						arrCyCtrl[arrCyNo.ElectValveName.CaDTCarryingVacuum].Cmd.bON:=TRUE;//负极叠片搬运真空破
						arrCyCtrl[arrCyNo.ElectValveName.CaDTCarryingVacuum].Cmd.bOFF:=FALSE;//负极叠片搬运真空破
						arrCyCtrl[arrCyNo.ElectValveName.CaCarryingVacuum2].Cmd.bON:=TRUE;//负极送片搬运真空破
						arrCyCtrl[arrCyNo.ElectValveName.CaCarryingVacuum2].Cmd.bOFF:=FALSE;//负极送片搬运真空破
						arrCyCtrl[arrCyNo.ElectValveName.CadeviationVacuum].Cmd.bON:=TRUE;//负极纠偏平台真空开
						arrCyCtrl[arrCyNo.ElectValveName.CadeviationVacuum].Cmd.bOFF:=FALSE;//负极纠偏平台真空开			
				
						  Mach_Control.Ca_b.Ca_DPCarryingFalg :=FALSE;//复位负极叠片搬运吸盘上有料标记
						//IF Mach_Control.Ca_b.Ca_CarryingFalg THEN
							Mach_Control.Ca_b.Ca_deviationFalg:=TRUE;//置位纠偏平台上有料标记
							Mach_Control.Ca_b.Ca_CarryingFalg:=FALSE;//复位负极送片搬运吸盘上有料标记
						//END_IF
						Par.stDT_date.Ca_MQ_Slice[8]:=Par.stDT_date.Ca_MQ_Slice[7];
			  END_IF
					
	END_IF	

		
	IF 	arrAxisCtrl[AxiseNo.VirAxisName.VirMain].Status.fActPos>=339   THEN//198
		    IF   NOT An_OverNGMark THEN	
					IF NOT Ca_Number    THEN
						CCD.Over.Start.iPhotoDo:=1;
					ELSE
						CCD.Over.Start.iPhotoDo:=2;
					END_IF
					CCD.Over.Finish.OverhandResult:=0;
					Mach_Control.DT_b.CDD_OverStart:=TRUE;
			  END_IF
					DP_Step3:=121;
					
	END_IF	
121:
	IF 	arrAxisCtrl[AxiseNo.VirAxisName.VirMain].Status.fActPos>=360 THEN//198
		 IF NOT An_OverNGMark THEN	
				arrCyCtrl[arrCyNo.ElectValveName.CaCarryingVacuum2].Cmd.bON:=FALSE;//负极送片搬运真空开
				arrCyCtrl[arrCyNo.ElectValveName.CaCarryingVacuum2].Cmd.bOFF:=TRUE;//负极送片搬运真空开
				arrCyCtrl[arrCyNo.ElectValveName.CaDTCarryingVacuum].Cmd.bON:=FALSE;//负极叠片搬运真空破
				arrCyCtrl[arrCyNo.ElectValveName.CaDTCarryingVacuum].Cmd.bOFF:=TRUE;//负极叠片搬运真空破
		   END_IF	
		DP_Step3:=6666;
	END_IF	
	
	
200://负极叠片，正极在取片位
		IF arrAxisCtrl[AxiseNo.VirAxisName.VirMain].Status.fActPos>=10  AND arrAxisCtrl[AxiseNo.VirAxisName.VirMain].Status.fActPos<=20 THEN//20240508 CF
			An_Step0:=10;//调用正极取片程序
			DP_Step3:=202;		
		END_IF
	
202:
	IF iAnCamInSel2=1 AND NOT An_OverNGMark  THEN
		arrCyCtrl[arrCyNo.ElectValveName.AnDTCarryingVacuum].Cmd.bON:=FALSE;//正极送片搬运真空开
		arrCyCtrl[arrCyNo.ElectValveName.AnDTCarryingVacuum].Cmd.bOFF:=TRUE;//正极送片搬运真空开
	END_IF
	
	//fbAnDTCarryingVacuum.Vacuumsel:=SEL(iAnCamInSel2=1,0,1)     ;//	正极叠片搬运真空开	
	IF arrAxisCtrl[AxiseNo.VirAxisName.VirMain].Status.fActPos>=235 THEN//复检提前
		IF Mach_Control.DT_b.DT_CCD_TwoModel THEN												
			CCD.AnRec.Finish.RectifyResult:=0;
			CCD.AnRec.Finish.RectifyX1:=0;
			CCD.AnRec.Finish.RectifyX2:=0;
			CCD.AnRec.Finish.RectifyY:=0;												
			Mach_Control.An_b.An_CCDStart :=TRUE;//启动CCD拍照
			CCD.AnRec.Start.iPhotoDo:=2;//第二次拍照	
		END_IF
		DP_Step3:=205;
	END_IF
205:			
	IF NOT DP_CheseCam  AND NOT  An_JumpRules[3]  AND NOT  An_JumpRules[6] AND NOT An_JumpRules[8] AND NOT An_JumpRules[10]    THEN
	
				IF arrAxisCtrl[AxiseNo.VirAxisName.VirMain].Status.fActPos>=250  AND arrAxisCtrl[AxiseNo.VirAxisName.VirMain].Status.fActPos<=255 THEN	
					        IF NOT An_OverNGMark THEN
										//fbAnCamInCarryingUpDown.bCamInExecute:=FALSE;//正极升解除耦合															
										//fbAnCamInCarryingWhirling.bCamInExecute:=FALSE;//正极旋转解除耦合			
										//Mach_Control.An_b.An_MainBelting:=FALSE;//正极搬运升降取极片中																					
										IF  NOT  Mach_Control.Ca_b.Ca_deviationFPOK  THEN    //负极放片纠偏太未在初始位置报警  
												Mach_Control.Ca_b.Error_tips[1]:=TRUE ;
										END_IF											
										IF  NOT  Mach_Control.An_b.An_deviationDPOK  THEN    //正极取片纠偏未完成报警
												Mach_Control.An_b.Error_tips[1]:=TRUE;
										END_IF			
										IF Mach_Control.An_b.An_deviationDPOK OR Mach_Control.U.EmptyRunMode OR	TRUE  THEN // 
											arrCyCtrl[arrCyNo.ElectValveName.AnDTCarryingVacuum].Cmd.bON:=FALSE;//正极叠片搬运真空开	
											arrCyCtrl[arrCyNo.ElectValveName.AnDTCarryingVacuum].Cmd.bOFF:=TRUE;//正极叠片搬运真空开		
											An_deviationDPOKFalg:=TRUE;	
										ELSE		
											arrCyCtrl[arrCyNo.ElectValveName.AnDTCarryingVacuum].Cmd.bON:=TRUE;//正极叠片搬运真空关					
											arrCyCtrl[arrCyNo.ElectValveName.AnDTCarryingVacuum].Cmd.bOFF:=FALSE;//正极叠片搬运真空关												
											fbAnCamInDTCarryingUpDown.bCamInExecute:=FALSE;	//正极叠片搬运升降凸轮解耦				
											IF NOT arrAxisCtrl[AxiseNo.AxisName.AnDTCarryingUpDown].Cmd.arrbRealPoint[4]    THEN
													arrAxisCtrl[AxiseNo.AxisName.AnDTCarryingUpDown].Cmd.iGoSetPos:=4;   //到等待位
											END_IF			
										END_IF	
										//IF NOT Mach_Control.An_b.JumpPiceReady THEN
											//An_Step0:=10;//调用正极取片程序	  20240509 CF
										//END_IF
										DP_Step3:=210;				
							 ELSE
							        DP_Step3:=210;	
				             END_IF
				 END_IF			 
	ELSE
									DP_Step3:=210;									
    END_IF

210:
	//打开或关闭真空，标记对应位置有料
	IF 	arrAxisCtrl[AxiseNo.VirAxisName.VirMain].Status.fActPos>=260 THEN//198
		  IF  NOT An_OverNGMark THEN
					CCD.Over.Start.iPliesNo:=UINT_TO_INT(Mach_Control.Ca_b.Ca_Quantited + Mach_Control.An_b.An_Quantited+1);
				    IF (CCD.Over.Start.iPliesNo MOD 2) <>1 OR CCD.Over.Start.iPliesNo=0 THEN
					   Mach_Control.DT_b.Error[69]:=TRUE;//负极对齐度拍照发送层数错误
				    END_IF					
					
					CCD.Over.Start.stPoleNo:=Par.stDT_date.Ca_MQ_Slice[8].stPoleNo;
							Mach_Control.Ca_b.Ca_Rectifydev_CS:=0;
					
							arrCyCtrl[arrCyNo.ElectValveName.CaCarryingVacuum2].Cmd.bON:=TRUE;//负极送片搬运真空关
							arrCyCtrl[arrCyNo.ElectValveName.CaCarryingVacuum2].Cmd.bOFF:=FALSE;//负极送片搬运真空关
							arrCyCtrl[arrCyNo.ElectValveName.CaDTCarryingVacuum].Cmd.bON:=TRUE;//负极叠片搬运直空关
							arrCyCtrl[arrCyNo.ElectValveName.CaDTCarryingVacuum].Cmd.bOFF:=FALSE;//负极叠片搬运直空关
							arrCyCtrl[arrCyNo.ElectValveName.CadeviationVacuum].Cmd.bON:=TRUE;//负极纠偏平台真空开	
							arrCyCtrl[arrCyNo.ElectValveName.CadeviationVacuum].Cmd.bOFF:=FALSE;//负极纠偏平台真空开		
							
							Mach_Control.Ca_b.Ca_DPCarryingFalg :=FALSE;//复位负极叠片搬运吸盘上有料标记
							//IF Mach_Control.Ca_b.Ca_CarryingFalg THEN
								Mach_Control.Ca_b.Ca_deviationFalg:=TRUE;//置位纠偏平台上有料标记
								Mach_Control.Ca_b.Ca_CarryingFalg:=FALSE;//复位负极送片搬运吸盘上有料标记
							//END_IF
							Par.stDT_date.Ca_MQ_Slice[8]:=Par.stDT_date.Ca_MQ_Slice[7];
							IF An_deviationDPOKFalg AND  iAnCamInSel2=1   THEN
									Par.stDT_date.An_MQ_Slice[2]:=Par.stDT_date.An_MQ_Slice[1];
									//IF Mach_Control.An_b.An_deviationFalg THEN
										Mach_Control.An_b.An_DPCarryingFalg :=TRUE;//复位正极叠片搬运吸盘上有料标记										
										Mach_Control.An_b.An_deviationFalg:=FALSE;//置位纠偏平台上有料标记	
									//END_IF										
									arrCyCtrl[arrCyNo.ElectValveName.AndeviationVacuum].Cmd.bOFF:=TRUE;//正极纠偏平台真空关
									arrCyCtrl[arrCyNo.ElectValveName.AndeviationVacuum].Cmd.bON:=FALSE;//正极纠偏平台真空关
									arrCyCtrl[arrCyNo.ElectValveName.AndeviationVacuumBark].Cmd.bON:=TRUE;//正极纠偏平台破真空开	
									arrCyCtrl[arrCyNo.ElectValveName.AndeviationVacuumBark].Cmd.bOFF:=FALSE;//正极纠偏平台破真空开	
							 END_IF			
							(*	
								ELSIF NOT   DP_CheseCam THEN								
									An_Step3:=10;//正极叠片搬运取纠偏台极片	
							*)																					
	        END_IF
				 
				 
	END_IF
	
	IF 	arrAxisCtrl[AxiseNo.VirAxisName.VirMain].Status.fActPos>=339 THEN//198
		  IF  NOT An_OverNGMark THEN
				IF NOT Ca_Number  THEN
					CCD.Over.Start.iPhotoDo:=1;
				ELSE
					CCD.Over.Start.iPhotoDo:=2;
				END_IF
				CCD.Over.Finish.OverhandResult:=0;
				Mach_Control.DT_b.CDD_OverStart:=TRUE;			
	       END_IF
				 
			IF NOT Ca_Number THEN
				DP_Step3:=211;					
			END_IF
	END_IF
	

211:
	IF 	arrAxisCtrl[AxiseNo.VirAxisName.VirMain].Status.fActPos>=360 THEN//198	
		 IF NOT An_OverNGMark THEN	
				arrCyCtrl[arrCyNo.ElectValveName.CaCarryingVacuum2].Cmd.bON:=FALSE;//负极送片搬运真空开
				arrCyCtrl[arrCyNo.ElectValveName.CaCarryingVacuum2].Cmd.bOFF:=TRUE;//负极送片搬运真空开
				arrCyCtrl[arrCyNo.ElectValveName.CaDTCarryingVacuum].Cmd.bON:=FALSE;//负极叠片搬运直空开
				arrCyCtrl[arrCyNo.ElectValveName.CaDTCarryingVacuum].Cmd.bOFF:=TRUE;//负极叠片搬运直空开
		END_IF		
		DP_Step3:=6666;					
	END_IF
			



		
300://正极叠片，负极在取片位			
	bStandbyStep1_3:=FALSE;
	bStandbyStep1_4:=FALSE;
	DP_Step3:=310; 		
310:	
	IF arrAxisCtrl[AxiseNo.VirAxisName.VirMain].Status.fActPos>=10  AND  arrAxisCtrl[AxiseNo.VirAxisName.VirMain].Status.fActPos<=245    THEN
		//正送片搬运极取片处理
		IF   arrAxisCtrl[AxiseNo.AxisName.CaCarryingUpDown2].Cmd.arrbRealPoint[4] AND 
			NOT Mach_Control.Ca_b.Ca_CarryingFalg    AND  ( Mach_Control.Ca_b.Ca_CacheBeltDLOK OR  Mach_Control.U.EmptyRunMode )  AND 
			NOT  Mach_Control.Ca_b.Ca_CacheBelting   AND NOT  bStandbyStep1_3 	 THEN
			Ca_Step0:=10;   //负极取流水线子程序
			bStandbyStep1_3:=TRUE;
		END_IF
	
		IF arrAxisCtrl[AxiseNo.AxisName.CaDTCarryingUpDown].Cmd.arrbRealPoint[4] AND 
			Mach_Control.Ca_b.Ca_deviationDPOK AND NOT Mach_Control.Ca_b.Ca_DPCarryingFalg AND  
			Mach_Control.Ca_b.Ca_deviationFalg AND  NOT  bStandbyStep1_4   
           AND   NOT Ca_OverNGMark THEN
			Ca_Step3:=10;     //负极取纠偏平台子程序
			bStandbyStep1_4:=TRUE;
		END_IF					
	ELSIF  arrAxisCtrl[AxiseNo.VirAxisName.VirMain].Status.fActPos>245  THEN
		    IF  NOT Ca_OverNGMark THEN
			      DP_Step3:=320; 
			ELSE	  
				  DP_Step3:=6666;	
			END_IF		  
	END_IF	
	
320://正极叠片，负极在取片位
   IF NOT Ca_OverNGMark THEN
		arrCyCtrl[arrCyNo.ElectValveName.AndeviationVacuum].Cmd.bON:=TRUE;//正极纠偏平台真空开			
		arrCyCtrl[arrCyNo.ElectValveName.AndeviationVacuum].Cmd.bOFF:=FALSE;//正极纠偏平台真空开		
	END_IF					
	IF 	arrAxisCtrl[AxiseNo.VirAxisName.VirMain].Status.fActPos>=260 THEN//198

		IF NOT Ca_OverNGMark THEN
				CCD.Over.Start.iPliesNo:=UINT_TO_INT(Mach_Control.Ca_b.Ca_Quantited + Mach_Control.An_b.An_Quantited+1);
				    IF (CCD.Over.Start.iPliesNo MOD 2) <>0 OR CCD.Over.Start.iPliesNo=0 THEN
					   Mach_Control.DT_b.Error[68]:=TRUE;//正极对齐度拍照发送层数错误
				    END_IF				
				
				CCD.Over.Start.stPoleNo:=Par.stDT_date.An_MQ_Slice[2].stPoleNo;
				Mach_Control.An_b.An_Rectifydev_CS:=0;				
		
				arrCyCtrl[arrCyNo.ElectValveName.AnCarryingVacuum].Cmd.bON:=FALSE;//正极送片搬运真空关
				arrCyCtrl[arrCyNo.ElectValveName.AnCarryingVacuum].Cmd.bOFF:=TRUE;//正极送片搬运真空关
				arrCyCtrl[arrCyNo.ElectValveName.AnCarryingVacuumBark].Cmd.bON:=TRUE;//正极送片搬运破真空开
				arrCyCtrl[arrCyNo.ElectValveName.AnCarryingVacuumBark].Cmd.bOFF:=FALSE;//正极送片搬运破真空开
				
				arrCyCtrl[arrCyNo.ElectValveName.AnDTCarryingVacuum].Cmd.bON:=TRUE;//正极送片搬运真空关
				arrCyCtrl[arrCyNo.ElectValveName.AnDTCarryingVacuum].Cmd.bOFF:=FALSE;//正极送片搬运真空关
				//arrCyCtrl[arrCyNo.ElectValveName.AnDTCarryingVacuumBark].Cmd.bON:=TRUE;//正极送片搬运破真空开
				//arrCyCtrl[arrCyNo.ElectValveName.AnDTCarryingVacuumBark].Cmd.bOFF:=FALSE;//正极送片搬运破真空开
				
				arrCyCtrl[arrCyNo.ElectValveName.AndeviationVacuum].Cmd.bON:=TRUE;//正极纠偏平台真空开		
				arrCyCtrl[arrCyNo.ElectValveName.AndeviationVacuum].Cmd.bOFF:=FALSE;//正极纠偏平台真空开		
				
				
				Mach_Control.An_b.An_DPCarryingFalg :=FALSE;//复位正极叠片搬运吸盘上有料标记
				//IF Mach_Control.An_b.An_CarryingFalg THEN
					Mach_Control.An_b.An_deviationFalg:=TRUE;//置位纠偏平台上有料标记
					Mach_Control.An_b.An_CarryingFalg:=FALSE;//复位正极送片搬运吸盘上有料标记
				//END_IF
				Par.stDT_date.An_MQ_Slice[1]:=Par.stDT_date.An_MQ_Slice[0];
	      END_IF				
	 END_IF

	IF 	arrAxisCtrl[AxiseNo.VirAxisName.VirMain].Status.fActPos>=339 THEN//198
		   IF NOT Ca_OverNGMark THEN
				IF NOT An_Number  THEN
					CCD.Over.Start.iPhotoDo:=1;
				ELSE
					CCD.Over.Start.iPhotoDo:=2;
				END_IF
				CCD.Over.Finish.OverhandResult:=0;
				Mach_Control.DT_b.CDD_OverStart:=TRUE;	
	       END_IF      
		  DP_Step3:=6666;	
	END_IF	
			

400:	//复检提前------//正极叠片，负极在叠片位
		IF arrAxisCtrl[AxiseNo.VirAxisName.VirMain].Status.fActPos>=10  AND arrAxisCtrl[AxiseNo.VirAxisName.VirMain].Status.fActPos<=20 THEN//20240508 CF																			
			Ca_Step0:=10;//调用负极取片程序       取片允许条件在子程序里
			DP_Step3:=402;
		END_IF

402:	
	//fbCaDTCarryingVacuum.Vacuumsel:= SEL(iCaCamInSel2=1 ,0,1)   ;//	负极叠片搬运真空开
	IF iCaCamInSel2=1 AND NOT Ca_OverNGMark THEN
		arrCyCtrl[arrCyNo.ElectValveName.CaDTCarryingVacuum].Cmd.bON:=FALSE;//负极叠台搬运真空开	
		arrCyCtrl[arrCyNo.ElectValveName.CaDTCarryingVacuum].Cmd.bOFF:=TRUE;//负极叠台搬运真空开		
	END_IF

	IF 	arrAxisCtrl[AxiseNo.VirAxisName.VirMain].Status.fActPos>=235 THEN//198
		IF Mach_Control.DT_b.DT_CCD_TwoModel THEN
				CCD.CaRec.Finish.RectifyX1:=0;
				CCD.CaRec.Finish.RectifyX2:=0;
				CCD.CaRec.Finish.RectifyY:=0;		
				CCD.CaRec.Finish.RectifyResult:=0;//拍照结果清零									
				Mach_Control.Ca_b.Ca_CCDStart :=TRUE;//启动CCD拍照
				CCD.CaRec.Start.iPhotoDo:=2;//启动CCD第二次拍照									
		END_IF
		DP_Step3:=405;
	END_IF
405:		
 
				IF arrAxisCtrl[AxiseNo.VirAxisName.VirMain].Status.fActPos>=250  AND arrAxisCtrl[AxiseNo.VirAxisName.VirMain].Status.fActPos<=255 THEN		
						  IF  NOT Ca_OverNGMark	  THEN															
										IF  NOT  Mach_Control.An_b.An_deviationFPOK  THEN    //正极放片纠偏太未在初始位置报警  
											  Mach_Control.An_b.Error_tips[2]:=TRUE ;
										END_IF
										
										IF  NOT  Mach_Control.Ca_b.Ca_deviationDPOK  THEN    //负极取片纠偏未完成报警
											  Mach_Control.Ca_b.Error_tips[2]:=TRUE ;
										END_IF		
								
										//正极叠片时平移到位后判断正极纠偏台是否允许放片
										IF Mach_Control.An_b.An_deviationFPOK OR Mach_Control.U.EmptyRunMode  THEN 
												An_deviationFPOKFalg:=TRUE;//正极纠偏平台允许放片标记
										ELSE									
											fbAnCamInCarryingUpDown.bCamInExecute:=FALSE;	//正极送片搬运升降凸轮解耦				
											IF NOT arrAxisCtrl[AxiseNo.AxisName.AnCarryingUpDown].Cmd.arrbRealPoint[4]    THEN
												arrAxisCtrl[AxiseNo.AxisName.AnCarryingUpDown].Cmd.iGoSetPos:=4;
											END_IF;				
										END_IF					
										IF Mach_Control.Ca_b.Ca_deviationDPOK OR Mach_Control.U.EmptyRunMode OR TRUE  THEN //  
											Ca_deviationDPOKFalg:=TRUE;	
											arrCyCtrl[arrCyNo.ElectValveName.CaDTCarryingVacuum].Cmd.bON:=FALSE;//负极叠片搬运真空开	
											arrCyCtrl[arrCyNo.ElectValveName.CaDTCarryingVacuum].Cmd.bOFF:=TRUE;//负极叠片搬运真空开		
										ELSE	
											//arrCyCtrl[arrCyNo.ElectValveName.CaDTCarryingVacuum].Cmd.bON:=FALSE;//负极叠片搬运真空开									
											fbCaCamInDTCarryingUpDown.bCamInExecute:=FALSE;	//负极叠片搬运升降凸轮解耦				
											IF NOT arrAxisCtrl[AxiseNo.AxisName.CaDTCarryingUpDown].Cmd.arrbRealPoint[4]    THEN
												arrAxisCtrl[AxiseNo.AxisName.CaDTCarryingUpDown].Cmd.iGoSetPos:=4;   //到等待位
											ELSE
												arrAxisCtrl[AxiseNo.AxisName.CaDTCarryingUpDown].Cmd.iGoSetPos:=0;   //到等待位
											END_IF;				
										END_IF			
											//Ca_Step0:=10;//调用负极取片程序       取片允许条件在子程序里 20240509 CF
											DP_Step3:=410;	
							ELSE
										   DP_Step3:=6666;			
							END_IF									
									
	           END_IF
	
(*	
	//判断是否允许负极送片搬运取料
	IF arrAxisCtrl[AxiseNo.VirAxisName.VirMain].Status.fActPos>=CamOutArgel  AND arrAxisCtrl[AxiseNo.VirAxisName.VirMain].Status.fActPos<=(CamOutArgel+5) THEN
		IF (Mach_Control.Ca_b.Ca_CacheBeltDLOK AND NOT fbCaCamInCarryingUpDown2OutCamFlge) OR Mach_Control.U.EmptyRunMode  THEN
			Mach_Control.Ca_b.Ca_CacheBelting:=TRUE;//f负极搬运升降取极片中	
			arrCyCtrl[arrCyNo.ElectValveName.CaCarryingVacuum2].Cmd.bON:=FALSE;//负极送片搬运真空开
			arrCyCtrl[arrCyNo.ElectValveName.CaCarryingVacuum2].Cmd.bOFF:=TRUE;//负极送片搬运真空开
		ELSE
			//arrCyCtrl[arrCyNo.ElectValveName.CaCarryingVacuum2].Cmd.bON:=FALSE;//负极送片搬运真空开
			fbCaCamInCarryingUpDown2.bCamInExecute:=FALSE;//负极升解除耦合
			Mach_Control.Ca_b.Ca_CacheBelting:=FALSE;
		END_IF								
	END_IF
	//解除负极搬运升降凸轮耦合标记
	fbCaCamInCarryingUpDown2OutCam_F_TRIG(CLK:=fbCaCamInCarryingUpDown2.bCamInExecute , Q=> );
	IF fbCaCamInCarryingUpDown2OutCam_F_TRIG.Q THEN
		fbCaCamInCarryingUpDown2OutCamFlge:=TRUE;//负极升降2凸轮解耦标记
	END_IF	
*)			
410:							
	//打开或关闭真空，标记对应位置有料
	IF 	arrAxisCtrl[AxiseNo.VirAxisName.VirMain].Status.fActPos>=260 THEN//198
		CCD.Over.Start.iPliesNo:=UINT_TO_INT(Mach_Control.Ca_b.Ca_Quantited + Mach_Control.An_b.An_Quantited+1);	
		IF (CCD.Over.Start.iPliesNo MOD 2) <>0 OR CCD.Over.Start.iPliesNo=0 THEN
		   Mach_Control.DT_b.Error[68]:=TRUE;//正极对齐度拍照发送层数错误
		END_IF	
	
		Mach_Control.An_b.An_Rectifydev_CS:=0;
			
					CCD.Over.Start.stPoleNo:=Par.stDT_date.An_MQ_Slice[2].stPoleNo;
				(*	
					arrCyCtrl[arrCyNo.ElectValveName.AnCarryingVacuum].Cmd.bOFF:=TRUE;//正极送片搬运真空关
					arrCyCtrl[arrCyNo.ElectValveName.AnCarryingVacuumBark].Cmd.bON:=TRUE;//正极送片搬运破真空开
					arrCyCtrl[arrCyNo.ElectValveName.AnDTCarryingVacuum].Cmd.bOFF:=TRUE;//正极叠片搬运真空关
					arrCyCtrl[arrCyNo.ElectValveName.AnDTCarryingVacuumBark].Cmd.bON:=TRUE;//正极叠片搬运破真空开
				*)	
					arrCyCtrl[arrCyNo.ElectValveName.AnCarryingVacuum].Cmd.bON:=FALSE;//正极送片搬运真空关
					arrCyCtrl[arrCyNo.ElectValveName.AnCarryingVacuum].Cmd.bOFF:=TRUE;//正极送片搬运真空关
					arrCyCtrl[arrCyNo.ElectValveName.AnCarryingVacuumBark].Cmd.bON:=TRUE;//正极送片搬运破真空开
					arrCyCtrl[arrCyNo.ElectValveName.AnCarryingVacuumBark].Cmd.bOFF:=FALSE;//正极送片搬运破真空开
					
					arrCyCtrl[arrCyNo.ElectValveName.AnDTCarryingVacuum].Cmd.bON:=TRUE;//正极送片搬运真空关
					arrCyCtrl[arrCyNo.ElectValveName.AnDTCarryingVacuum].Cmd.bOFF:=FALSE;//正极送片搬运真空关
					//arrCyCtrl[arrCyNo.ElectValveName.AnDTCarryingVacuumBark].Cmd.bON:=TRUE;//正极送片搬运破真空开
				//	arrCyCtrl[arrCyNo.ElectValveName.AnDTCarryingVacuumBark].Cmd.bOFF:=FALSE;//正极送片搬运破真空开	
					
					arrCyCtrl[arrCyNo.ElectValveName.AndeviationVacuum].Cmd.bON:=TRUE;//正极纠偏平台真空开	
					arrCyCtrl[arrCyNo.ElectValveName.AndeviationVacuum].Cmd.bOFF:=FALSE;//正极纠偏平台真空开	
			
					Mach_Control.An_b.An_DPCarryingFalg :=FALSE;//复位正极叠片搬运吸盘上有料标记
					//IF Mach_Control.An_b.An_CarryingFalg THEN
						Mach_Control.An_b.An_deviationFalg:=TRUE;//置位纠偏平台上有料标记
						Mach_Control.An_b.An_CarryingFalg:=FALSE;//复位正极送片搬运吸盘上有料标记
					//END_IF
					
					Par.stDT_date.An_MQ_Slice[1]:=Par.stDT_date.An_MQ_Slice[0];
					
					(*
					IF (Mach_Control.Ca_b.Ca_CacheBelting AND NOT fbCaCamInCarryingUpDown2OutCamFlge) OR Mach_Control.U.EmptyRunMode  THEN
						Mach_Control.Ca_b.Ca_CarryingFalg:=TRUE;//复位负极送片搬运吸盘上有料标记
						Par.stDT_date.Ca_MQ_Slice[7]:=Par.stDT_date.Ca_MQ_Slice[6];
					END_IF*)
					
					
					arrAxisCtrl[AxiseNo.AxisName.CaCarryingUpDown2].Cmd.bStop:=FALSE;
				


		//判断负极纠偏台是否允许取料
		IF Ca_deviationDPOKFalg AND NOT DP_CheseCam AND iCaCamInSel2=1 AND   NOT Ca_OverNGMark	 THEN		
			arrCyCtrl[arrCyNo.ElectValveName.CaDTCarryingVacuum].Cmd.bON:=FALSE;//负极叠台搬运真空开	
			arrCyCtrl[arrCyNo.ElectValveName.CaDTCarryingVacuum].Cmd.bOFF:=TRUE;//负极叠台搬运真空开	
			arrCyCtrl[arrCyNo.ElectValveName.CadeviationVacuum].Cmd.bOFF:=TRUE;//负极纠偏平台真空关
			arrCyCtrl[arrCyNo.ElectValveName.CadeviationVacuum].Cmd.bON:=FALSE;//负极纠偏平台真空关
			arrCyCtrl[arrCyNo.ElectValveName.CadeviationVacuumBark].Cmd.bON:=TRUE;//负极纠偏平台破真空开	
			arrCyCtrl[arrCyNo.ElectValveName.CadeviationVacuumBark].Cmd.bOFF:=FALSE;//负极纠偏平台破真空开		
			//IF 	Mach_Control.Ca_b.Ca_deviationFalg THEN				
				Mach_Control.Ca_b.Ca_DPCarryingFalg :=TRUE;//置位负极叠片搬运吸盘上有料标记			
				Mach_Control.Ca_b.Ca_deviationFalg:=FALSE;//复位负极纠偏平台上有料标记	
			//END_IF			
			Par.stDT_date.Ca_MQ_Slice[9]:=Par.stDT_date.Ca_MQ_Slice[8];
		(*	
		ELSE   
			Ca_Step3:=10;//负极叠片搬运取纠偏台极片	
		*)	   
		END_IF									

		//判断正极纠偏台是否允许放料
		IF  NOT Ca_OverNGMark	 THEN		
				IF An_deviationFPOKFalg THEN			
					arrCyCtrl[arrCyNo.ElectValveName.AnCarryingVacuumBark].Cmd.bON:=TRUE;//正极送片搬运真空关
					arrCyCtrl[arrCyNo.ElectValveName.AnCarryingVacuumBark].Cmd.bOFF:=FALSE;//正极送片搬运破真空开
					arrCyCtrl[arrCyNo.ElectValveName.AndeviationVacuum].Cmd.bON:=TRUE;//正极纠偏平台真空开		
					arrCyCtrl[arrCyNo.ElectValveName.AndeviationVacuum].Cmd.bOFF:=FALSE;//正极纠偏平台真空开	
					//IF Mach_Control.An_b.An_CarryingFalg THEN	
						Mach_Control.An_b.An_deviationFalg:=TRUE;//置位正极纠偏平台上有料标记
						Mach_Control.An_b.An_CarryingFalg:=FALSE;//复位正极送片搬运吸盘上有料标记						
					//END_IF			
					Par.stDT_date.An_MQ_Slice[1]:=Par.stDT_date.An_MQ_Slice[0];//送片机械手传送至纠偏平台
					ELSE   
						An_Step1:=10;//正极送片搬运放片到纠偏台			   
					END_IF
			END_IF 
	END_IF

	IF 	arrAxisCtrl[AxiseNo.VirAxisName.VirMain].Status.fActPos>=339 THEN//198
		 IF NOT Ca_OverNGMark THEN
				IF NOT An_Number THEN
					CCD.Over.Start.iPhotoDo:=1;
				ELSE
					CCD.Over.Start.iPhotoDo:=2;
				END_IF
				CCD.Over.Finish.OverhandResult:=0;
				Mach_Control.DT_b.CDD_OverStart:=TRUE;	
	    END_IF
			
		IF NOT An_Number THEN
			DP_Step3:=6666;					
		END_IF

	
	END_IF
	

END_CASE



//判断主轴是否完成
CASE  DP_Step4 OF
100://叠负极主轴定位完成判断	
		//叠负极主轴在当前周期220度之前对齐度NG为上一片结果
      IF (((arrAxisCtrl[AxiseNo.VirAxisName.VirMain].Status.fActPos>10 AND  arrAxisCtrl[AxiseNo.VirAxisName.VirMain].Status.fActPos<230) AND 
           (CCD.Over.Finish.OverhandResult=2 OR  CCD.Over.Finish.OverhandResult=3 OR CCD.Over.Finish.OverhandResult=4 ) ) OR
		  (arrAxisCtrl[AxiseNo.VirAxisName.VirMain].Status.fActPos>=230 AND  arrAxisCtrl[AxiseNo.VirAxisName.VirMain].Status.fActPos<235 AND 
           CCD.Over.Finish.OverhandResult=0  ))  AND
           NOT Mach_Control.DT_b.DT_Overhang AND  NOT  Mach_Control.U.EmptyRunMode AND NOT Mach_Control.DT_b.DT_Sheetkick AND  
           Mach_Control.Ca_b.Ca_Quantited>0  AND NOT Ca_OverNGMark AND NOT OversequelNG AND NOT Bnt_Blueflaging THEN
		  An_OverNGMark:=TRUE;//上一片正极对齐度NG标记
	  END_IF

	  
	 IF  arrAxisCtrl[AxiseNo.VirAxisName.VirMain].Status.fActPos>240  THEN 
	      Ca_OverNGMark:=FALSE;
	  END_IF
	   
	IF arrAxis[AxiseNo.VirAxisName.VirMain].NcToPlc.SetPos=360 AND  arrAxis[AxiseNo.VirAxisName.VirMain].Status.NotMoving  THEN
		//如果，叠片搬运掉片报警就不计数		
		IF NOT Ca_Number AND NOT An_OverNGMark THEN
						Mach_Control.Ca_b.Ca_Quantited:=Mach_Control.Ca_b.Ca_Quantited+1;
						DPcount:=DPcount+1;
						IF Mach_Control.U.EmptyRunMode THEN
							Mach_Control.Ca_b.Ca_EmptyRunKDQuantited:=Mach_Control.Ca_b.Ca_EmptyRunKDQuantited +1;
						//			ELSE
						//				Mach_Control.Ca_b.Ca_EmptyRunKDQuantited:=0;
						END_IF
						Par.stDT_date.YD_JS_L:=Par.stDT_date.YD_JS_L+1;
						Par.stDT_date.YD_ferrJS:=Par.stDT_date.YD_ferrJS+1;
						Mach_Control.Ca_b.Ca_CCD_amount:=0;
							//叠台升降轴下降
							IF NOT Mach_Control.U.EmptyRunMode  THEN
								arrAxisCtrl[AxiseNo.AxisName.DTUpDown].Cmd.fPosition_of_Rel:=-(Par.stDT_date.Ca_Thickness+Par.stDT_date.SEPTA_Thickness+Par.stDT_date.Pole_ThicknessCom);
							ELSE
								arrAxisCtrl[AxiseNo.AxisName.DTUpDown].Cmd.fPosition_of_Rel:=-Par.stDT_date.SEPTA_Thickness;
							END_IF
							IF Mach_Control.Ca_b.Ca_Quantited + Mach_Control.An_b.An_Quantited>3 THEN
								arrAxisPar[AxiseNo.AxisName.DTUpDown].fVelocity_of_Rel:=100;
								arrAxisCtrl[AxiseNo.AxisName.DTUpDown].Cmd.bMoveRel:=TRUE;
							END_IF
		END_IF
		Mach_Control.An_b.An_CCDStart :=FALSE;//启动CCD拍照						
		DP_Step1:=100;//解除耦合，主轴回零子程序
	    

		IF Mach_Control.DT_b.SinStepMode THEN//单步调试模式
			DP_SinStepe:=TRUE;
		ELSE
			DP_SinStepe:=FALSE;	
		END_IF
		
		//DP_Step0:=0;
		Ca_AlarmTON[11].IN:=FALSE;
		IF Ca_Number  OR An_OverNGMark THEN
			DP_Step6:=6666;
		ELSIF Mach_Control.DT_b.DT_Overhang THEN
			DP_Step6:=102;
		ELSE
			DP_Step6:=101;
		END_IF	
		DP_Step4:=110;
        DPtime:=10;	
	END_IF;	
110:
	IF ((*Ca_deviationFPOKFalg OR*) Ca_Step1=6666 OR Ca_Step1=0) AND ((*An_deviationDPOKFalg OR *)An_Step3=6666 OR An_Step3=0)  
		AND ((An_Step0=6666 OR An_Step0=0) OR Mach_Control.An_b.An_Quantited=Par.stDT_date.An_Quantity )  THEN         
		DP_Step4:=6666;
			IF   NOT An_OverNGMark THEN
	        	DP_Step0:=0;
				DPtime:=11;	
		       Ca_deviationFPOKFalg:=FALSE;
		       An_deviationDPOKFalg:=FALSE;  
			ELSE   
			    DP_Step0:=10;
		     	An_OverNGStep:=1000;	//踢正极对齐度NG片
				 CCD.Over.Finish.OverhandResult:=0;	
	       END_IF;				
	END_IF



		
200:	//叠正极主轴定位完成判断
	  //叠正极主轴在当前周期220度之前对齐度NG为上一片结果
	   IF (((arrAxisCtrl[AxiseNo.VirAxisName.VirMain].Status.fActPos>10 AND  arrAxisCtrl[AxiseNo.VirAxisName.VirMain].Status.fActPos<230) AND 
           (CCD.Over.Finish.OverhandResult=2 OR  CCD.Over.Finish.OverhandResult=3 OR CCD.Over.Finish.OverhandResult=4 )) OR
           (arrAxisCtrl[AxiseNo.VirAxisName.VirMain].Status.fActPos>=230 AND  arrAxisCtrl[AxiseNo.VirAxisName.VirMain].Status.fActPos<235 AND 
            CCD.Over.Finish.OverhandResult=0))  AND     
           NOT Mach_Control.DT_b.DT_Overhang AND NOT  Mach_Control.U.EmptyRunMode  AND NOT Mach_Control.DT_b.DT_Sheetkick AND
           Mach_Control.Ca_b.Ca_Quantited>0  AND NOT An_OverNGMark AND NOT OversequelNG AND NOT Bnt_Blueflaging THEN
		  Ca_OverNGMark:=TRUE;//上一片负极对齐度NG标记
	  END_IF
	
	 	 IF  arrAxisCtrl[AxiseNo.VirAxisName.VirMain].Status.fActPos>240 THEN 
	      An_OverNGMark:=FALSE;
	  END_IF 
	  
	
	IF arrAxis[AxiseNo.VirAxisName.VirMain].NcToPlc.SetPos=360 AND  arrAxis[AxiseNo.VirAxisName.VirMain].Status.NotMoving  THEN
		//如果，叠片搬运掉片报警就不计数				
		IF NOT An_Number AND NOT Ca_OverNGMark THEN
						Mach_Control.An_b.An_Quantited:=Mach_Control.An_b.An_Quantited+1;
						DPcount:=DPcount+1;			
						IF Mach_Control.U.EmptyRunMode THEN
							Mach_Control.An_b.An_EmptyRunKDQuantited:=Mach_Control.An_b.An_EmptyRunKDQuantited +1;
						//			ELSE
						//				Mach_Control.An_b.An_EmptyRunKDQuantited:=0;
						END_IF
						Par.stDT_date.YD_JS_R:=Par.stDT_date.YD_JS_R+1;
						Mach_Control.An_b.An_CCD_amount:=0;
						//叠台升降轴下降
						IF NOT Mach_Control.U.EmptyRunMode  THEN
								arrAxisCtrl[AxiseNo.AxisName.DTUpDown].Cmd.fPosition_of_Rel:=-(Par.stDT_date.An_Thickness+Par.stDT_date.SEPTA_Thickness+Par.stDT_date.Pole_ThicknessCom);
						ELSE
								arrAxisCtrl[AxiseNo.AxisName.DTUpDown].Cmd.fPosition_of_Rel:=-Par.stDT_date.SEPTA_Thickness;
						END_IF
						IF Mach_Control.Ca_b.Ca_Quantited + Mach_Control.An_b.An_Quantited>3 THEN
								arrAxisPar[AxiseNo.AxisName.DTUpDown].fVelocity_of_Rel:=100;
								arrAxisCtrl[AxiseNo.AxisName.DTUpDown].Cmd.bMoveRel:=TRUE;
						END_IF	
		END_IF
		Mach_Control.Ca_b.Ca_CCDStart :=FALSE;//启动CCD拍照			
		DP_Step1:=100;//解除耦合，主轴回零	
        
		(*
		IF  (Mach_Control.Ca_b.Ca_CacheBelting AND NOT fbCaCamInCarryingUpDown2OutCamFlge) OR Mach_Control.U.EmptyRunMode  THEN
			Par.stDT_date.Ca_betlCount.5:=FALSE;//复位负极流水线极片标记
			Mach_Control.Ca_b.Ca_CacheBelting:=FALSE;
		END_IF	*)
	
						
		arrCyCtrl[arrCyNo.ElectValveName.CadeviationVacuumBark].Cmd.bOFF:=TRUE;//负极纠偏平台破真空关	
		IF Mach_Control.DT_b.SinStepMode THEN//单步调试模式
			DP_SinStepe:=TRUE;
		ELSE
			DP_SinStepe:=FALSE;	
		END_IF							
		//DP_Step0:=0;
		An_AlarmTON[11].IN:=FALSE;
		IF An_Number OR Ca_OverNGMark THEN
			  DP_Step7:=6666;
		ELSIF  Mach_Control.DT_b.DT_Overhang THEN
			  DP_Step7:=202;
		ELSE
			  DP_Step7:=201;
		END_IF
		DP_Step4:=210;	
		DPtime:=20;	
		(*	
			IF  Mach_Control.DT_b.DT_Overhang AND NOT An_Number THEN
				  DP_Step7:=202;
			ELSIF An_Number THEN
				  DP_Step7:=6666;
			ELSE
				  DP_Step7:=201;
			END_IF
			DP_Step4:=6666;	
		*)
	END_IF;	
210:
	IF ((*An_deviationFPOKFalg OR *)An_Step1=6666 OR An_Step1=0) AND ((*Ca_deviationDPOKFalg OR *)Ca_Step3=6666 OR Ca_Step3=0) 
	AND (Ca_Step0=6666 OR Ca_Step0=0) THEN       
          	DP_Step4:=6666;
          IF NOT Ca_OverNGMark THEN
				DP_Step0:=0;
				DPtime:=21;	
				An_deviationFPOKFalg:=FALSE;
				Ca_deviationDPOKFalg:=FALSE; 
			ELSE	
			    DP_Step0:=20;
		     	Ca_OverNGStep:=1000;	//踢负极对齐度NG片
                CCD.Over.Finish.OverhandResult:=0;	
          END_IF
			
	END_IF

			
END_CASE



//观察NG片用，发现问题后删除
IF Ca_NGTest1.Q THEN
	Ca_NG:=Ca_NG+1;
END_IF


CASE  DP_Step5 OF
100://判断主轴运行时负极叠片搬运升降真空报警
	IF arrAxisCtrl[AxiseNo.VirAxisName.VirMain].Status.fActPos>0 AND arrAxisCtrl[AxiseNo.VirAxisName.VirMain].Status.fActPos<235 THEN
		IF Ca_Number OR An_OverNGMark  THEN	
			IF Ca_Number THEN
				AnOverNGcount:=0; 
				arrCyCtrl[arrCyNo.ElectValveName.CaDTCarryingVacuum].Cmd.bON:=TRUE;//负极叠片搬运破真空开	
				arrCyCtrl[arrCyNo.ElectValveName.CaDTCarryingVacuum].Cmd.bOFF:=FALSE;//负极叠片搬运破真空开	
			END_IF	
				DP_Step5:=110;
		END_IF
		Ca_NGTest1(CLK:=(CCD.CaRec.Finish.RectifyResult=2) , Q=> );
	ELSE
		AnOverNGcount:=0; 
		DP_Step5:=6666;
	END_IF

110://叠负极主轴220度之前有对齐度NG, 负极送片搬运升降、负极叠台搬运升降、右压刀开合、右压刀升降、正极叠台搬运升降轴解耦  ,踢掉上一片正极
	fbCaCamInDTCarryingUpDown.bCamInExecute:=FALSE;//负极叠片搬运升降
	fbCamInLeftYDUpDown.bCamInExecute:=FALSE;//左压刀升降
	fbCamInLeftYDLine.bCamInExecute:=FALSE;//左压刀开合
	IF  An_OverNGMark THEN
		fbCaCamInCarryingUpDown2.bCamInExecute:=FALSE;//负极s送片搬运升降
		fbAnCamInDTCarryingUpDown.bCamInExecute:=FALSE;//正极叠片搬运升降
		IF NOT Mach_Control.An_b.An_DPCarryingFalg THEN
			arrCyCtrl[arrCyNo.ElectValveName.AnDTCarryingVacuum].Cmd.bON:=TRUE;//正极叠片搬运真空真空关
			arrCyCtrl[arrCyNo.ElectValveName.AnDTCarryingVacuum].Cmd.bOFF:=FALSE;//正极叠片搬运真空真空关
		END_IF	
	END_IF
	 
	IF NOT  fbCaCamInDTCarryingUpDown.bCamInExecute AND NOT fbCamInLeftYDUpDown.bCamInExecute AND NOT  fbCamInLeftYDLine.bCamInExecute AND 
        (( NOT  fbCaCamInCarryingUpDown2.bCamInExecute AND NOT  fbAnCamInDTCarryingUpDown.bCamInExecute ) OR NOT An_OverNGMark )   THEN
	       IF Ca_Number THEN
				arrCyCtrl[arrCyNo.ElectValveName.CaDTCarryingVacuum].Cmd.bON:=FALSE;//负极叠片搬运真空开
				arrCyCtrl[arrCyNo.ElectValveName.CaDTCarryingVacuum].Cmd.bOFF:=TRUE;//负极叠片搬运真空开
			END_IF	
			DP_Step5:=120;
	END_IF

120:
	arrAxisCtrl[AxiseNo.AxisName.CaDTCarryingUpDown].Cmd.bGearOut:=TRUE;
	arrAxisCtrl[AxiseNo.AxisName.LeftYDLine].Cmd.bGearOut:=TRUE;
	arrAxisCtrl[AxiseNo.AxisName.LeftYDUpDown].Cmd.bGearOut:=TRUE;
	IF  An_OverNGMark THEN
		arrAxisCtrl[AxiseNo.AxisName.CaCarryingUpDown2].Cmd.bGearOut:=TRUE;
		arrAxisCtrl[AxiseNo.AxisName.AnDTCarryingUpDown].Cmd.bGearOut:=TRUE;
	END_IF
	IF NOT arrAxisCtrl[AxiseNo.AxisName.CaDTCarryingUpDown].Status.Coupled AND NOT arrAxisCtrl[AxiseNo.AxisName.LeftYDLine].Status.Coupled AND 
       NOT arrAxisCtrl[AxiseNo.AxisName.LeftYDUpDown].Status.Coupled  AND 
         (( NOT arrAxisCtrl[AxiseNo.AxisName.CaCarryingUpDown2].Status.Coupled  AND NOT  arrAxisCtrl[AxiseNo.AxisName.AnDTCarryingUpDown].Status.Coupled )  OR NOT An_OverNGMark ) THEN
		arrAxisCtrl[AxiseNo.AxisName.CaDTCarryingUpDown].Cmd.bGearOut:=FALSE;
		arrAxisCtrl[AxiseNo.AxisName.LeftYDLine].Cmd.bGearOut:=FALSE;
		arrAxisCtrl[AxiseNo.AxisName.LeftYDUpDown].Cmd.bGearOut:=FALSE;
		IF  An_OverNGMark THEN
			arrAxisCtrl[AxiseNo.AxisName.CaCarryingUpDown2].Cmd.bGearOut:=FALSE;
			arrAxisCtrl[AxiseNo.AxisName.AnDTCarryingUpDown].Cmd.bGearOut:=FALSE;
		END_IF
		DP_Step5:=130;
	END_IF

130:
	IF arrAxisCtrl[AxiseNo.AxisName.CaDTCarryingUpDown].Status.Homed AND arrAxisCtrl[AxiseNo.AxisName.CaDTCarryingUpDown].Status.NoMoving AND 
		NOT arrAxisCtrl[AxiseNo.AxisName.CaDTCarryingUpDown].Status.Error THEN
		IF arrAxisCtrl[AxiseNo.AxisName.CaDTCarryingUpDown].Cmd.arrbRealPoint[4] THEN
			  IF Ca_Number THEN
					arrCyCtrl[arrCyNo.ElectValveName.CaDTCarryingVacuum].Cmd.bON:=FALSE;//负极叠片搬运真空开
					arrCyCtrl[arrCyNo.ElectValveName.CaDTCarryingVacuum].Cmd.bOFF:=TRUE;//负极叠片搬运真空开
			  END_IF		
			arrAxisCtrl[AxiseNo.AxisName.CaDTCarryingUpDown].Cmd.iGoSetPos:=0;
		ELSE
			arrAxisCtrl[AxiseNo.AxisName.CaDTCarryingUpDown].Cmd.iGoSetPos:=4;//负极叠片升降移动至等待高度
		END_IF
	
     IF An_OverNGMark THEN
					IF arrAxisCtrl[AxiseNo.AxisName.CaCarryingUpDown2].Status.Homed AND arrAxisCtrl[AxiseNo.AxisName.CaCarryingUpDown2].Status.NoMoving AND 
					NOT arrAxisCtrl[AxiseNo.AxisName.CaCarryingUpDown2].Status.Error THEN
							IF arrAxisCtrl[AxiseNo.AxisName.CaCarryingUpDown2].Cmd.arrbRealPoint[4] THEN
								arrAxisCtrl[AxiseNo.AxisName.CaCarryingUpDown2].Cmd.iGoSetPos:=0;
							ELSE
								arrAxisCtrl[AxiseNo.AxisName.CaCarryingUpDown2].Cmd.iGoSetPos:=4;//负极送片升降移动至等待高度
							END_IF	
					 END_IF
					 
					IF arrAxisCtrl[AxiseNo.AxisName.AnDTCarryingUpDown].Status.Homed AND arrAxisCtrl[AxiseNo.AxisName.AnDTCarryingUpDown].Status.NoMoving AND 
					NOT arrAxisCtrl[AxiseNo.AxisName.AnDTCarryingUpDown].Status.Error THEN
							IF arrAxisCtrl[AxiseNo.AxisName.AnDTCarryingUpDown].Cmd.arrbRealPoint[4] THEN
								arrAxisCtrl[AxiseNo.AxisName.AnDTCarryingUpDown].Cmd.iGoSetPos:=0;
							ELSE
								arrAxisCtrl[AxiseNo.AxisName.AnDTCarryingUpDown].Cmd.iGoSetPos:=4;//正极叠片升降移动至等待高度
							END_IF		
					END_IF
		END_IF			
		
		IF arrAxisCtrl[AxiseNo.AxisName.CaDTCarryingUpDown].Cmd.arrbRealPoint[4]  AND
			( (arrAxisCtrl[AxiseNo.AxisName.CaCarryingUpDown2].Cmd.arrbRealPoint[4]  AND arrAxisCtrl[AxiseNo.AxisName.AnDTCarryingUpDown].Cmd.arrbRealPoint[4]) OR NOT An_OverNGMark ) THEN
      		DP_Step5:=6666;
		END_IF
	END_IF







200://判断主轴运行时正极叠片搬运升降真空报警
	IF arrAxisCtrl[AxiseNo.VirAxisName.VirMain].Status.fActPos>0 AND arrAxisCtrl[AxiseNo.VirAxisName.VirMain].Status.fActPos<235 THEN
		IF An_Number OR Ca_OverNGMark THEN	
			IF An_Number THEN
				CaOverNGcount:=0;
		    //	arrCyCtrl[arrCyNo.ElectValveName.AnDTCarryingVacuumBark].Cmd.bON:=TRUE;//正极叠片搬运破真空开	
				arrCyCtrl[arrCyNo.ElectValveName.AnDTCarryingVacuum].Cmd.bON:=TRUE;//正极叠片搬运真空真空关
			    arrCyCtrl[arrCyNo.ElectValveName.AnDTCarryingVacuum].Cmd.bOFF:=FALSE;//正极叠片搬运真空真空关
			END_IF
			DP_Step5:=210;
		END_IF
	ELSE
		CaOverNGcount:=0; 
		DP_Step5:=6666;
	END_IF

210://叠正极主轴220度之前有对齐度NG, 正极送片搬运升降、正极叠台搬运升降、右压刀开合、右压刀升降、负极叠台搬运升降轴解耦  ,踢掉上一片负极
	fbAnCamInDTCarryingUpDown.bCamInExecute:=FALSE;//正极叠片搬运升降
	fbCamInRightYDUpDown.bCamInExecute:=FALSE;//右压刀升降
	fbCamInRightYDLine.bCamInExecute:=FALSE;//右压刀开会
	IF Ca_OverNGMark THEN
		fbAnCamInCarryingUpDown.bCamInExecute:=FALSE;//正极送片搬运升降
	    fbCaCamInDTCarryingUpDown.bCamInExecute:=FALSE;//负极叠片搬运升降
		IF NOT Mach_Control.Ca_b.Ca_DPCarryingFalg THEN
			arrCyCtrl[arrCyNo.ElectValveName.CaDTCarryingVacuum].Cmd.bON:=TRUE;//负极叠台搬运真空开	
			arrCyCtrl[arrCyNo.ElectValveName.CaDTCarryingVacuum].Cmd.bOFF:=FALSE;//负极叠台搬运真空开			
		END_IF	
	END_IF
	
	IF NOT fbAnCamInDTCarryingUpDown.bCamInExecute AND NOT fbCamInRightYDUpDown.bCamInExecute AND NOT fbCamInRightYDLine.bCamInExecute AND 
       (( NOT fbAnCamInCarryingUpDown.bCamInExecute AND NOT  fbCaCamInDTCarryingUpDown.bCamInExecute) OR NOT Ca_OverNGMark)  THEN
		IF An_Number THEN 
      		//arrCyCtrl[arrCyNo.ElectValveName.AnDTCarryingVacuumBark].Cmd.bON:=FALSE;//正极叠片搬运破真空关	
				arrCyCtrl[arrCyNo.ElectValveName.AnDTCarryingVacuum].Cmd.bON:=TRUE;//正极叠片搬运真空真空关
			    arrCyCtrl[arrCyNo.ElectValveName.AnDTCarryingVacuum].Cmd.bOFF:=FALSE;//正极叠片搬运真空真空关			
		END_IF
		DP_Step5:=220;
	END_IF
220:
	arrAxisCtrl[AxiseNo.AxisName.AnDTCarryingUpDown].Cmd.bGearOut:=TRUE;
	arrAxisCtrl[AxiseNo.AxisName.RightYDLine].Cmd.bGearOut:=TRUE;
	arrAxisCtrl[AxiseNo.AxisName.RightYDUpDown].Cmd.bGearOut:=TRUE;
	IF Ca_OverNGMark THEN
		arrAxisCtrl[AxiseNo.AxisName.AnCarryingUpDown].Cmd.bGearOut:=TRUE;
	   arrAxisCtrl[AxiseNo.AxisName.CaDTCarryingUpDown].Cmd.bGearOut:=TRUE;
	END_IF
	IF NOT arrAxisCtrl[AxiseNo.AxisName.AnDTCarryingUpDown].Status.Coupled AND NOT arrAxisCtrl[AxiseNo.AxisName.RightYDLine].Status.Coupled AND
		NOT arrAxisCtrl[AxiseNo.AxisName.RightYDUpDown].Status.Coupled  AND
      (( NOT arrAxisCtrl[AxiseNo.AxisName.AnCarryingUpDown].Status.Coupled AND NOT arrAxisCtrl[AxiseNo.AxisName.CaDTCarryingUpDown].Status.Coupled) OR NOT Ca_OverNGMark) THEN
		arrAxisCtrl[AxiseNo.AxisName.AnDTCarryingUpDown].Cmd.bGearOut:=FALSE;
		arrAxisCtrl[AxiseNo.AxisName.RightYDLine].Cmd.bGearOut:=FALSE;
		arrAxisCtrl[AxiseNo.AxisName.RightYDUpDown].Cmd.bGearOut:=FALSE;
		IF Ca_OverNGMark THEN
			arrAxisCtrl[AxiseNo.AxisName.AnCarryingUpDown].Cmd.bGearOut:=FALSE;
		    arrAxisCtrl[AxiseNo.AxisName.CaDTCarryingUpDown].Cmd.bGearOut:=FALSE;			
		END_IF
		DP_Step5:=230;
	END_IF

230:
	IF arrAxisCtrl[AxiseNo.AxisName.AnDTCarryingUpDown].Status.Homed AND arrAxisCtrl[AxiseNo.AxisName.AnDTCarryingUpDown].Status.NoMoving AND 
	NOT arrAxisCtrl[AxiseNo.AxisName.AnDTCarryingUpDown].Status.Error THEN
		IF arrAxisCtrl[AxiseNo.AxisName.AnDTCarryingUpDown].Cmd.arrbRealPoint[4] THEN
			arrAxisCtrl[AxiseNo.AxisName.AnDTCarryingUpDown].Cmd.iGoSetPos:=0;
		ELSE
			arrAxisCtrl[AxiseNo.AxisName.AnDTCarryingUpDown].Cmd.iGoSetPos:=4;//正极叠片升降移动至等待高度
		END_IF
	END_IF
	
	IF Ca_OverNGMark THEN
		IF arrAxisCtrl[AxiseNo.AxisName.AnCarryingUpDown].Status.Homed AND arrAxisCtrl[AxiseNo.AxisName.AnCarryingUpDown].Status.NoMoving AND 
	        NOT arrAxisCtrl[AxiseNo.AxisName.AnCarryingUpDown].Status.Error THEN
				IF arrAxisCtrl[AxiseNo.AxisName.AnCarryingUpDown].Cmd.arrbRealPoint[4] THEN
					arrAxisCtrl[AxiseNo.AxisName.AnCarryingUpDown].Cmd.iGoSetPos:=0;
				ELSE
					arrAxisCtrl[AxiseNo.AxisName.AnCarryingUpDown].Cmd.iGoSetPos:=4;//正极送片升降移动至等待高度
				END_IF
    	END_IF	
	
			IF arrAxisCtrl[AxiseNo.AxisName.CaDTCarryingUpDown].Status.Homed AND arrAxisCtrl[AxiseNo.AxisName.CaDTCarryingUpDown].Status.NoMoving AND 
	            NOT arrAxisCtrl[AxiseNo.AxisName.CaDTCarryingUpDown].Status.Error THEN
				IF arrAxisCtrl[AxiseNo.AxisName.CaDTCarryingUpDown].Cmd.arrbRealPoint[4] THEN
					arrAxisCtrl[AxiseNo.AxisName.CaDTCarryingUpDown].Cmd.iGoSetPos:=0;
				ELSE
					arrAxisCtrl[AxiseNo.AxisName.CaDTCarryingUpDown].Cmd.iGoSetPos:=4;//负极叠片升降移动至等待高度
				END_IF
    	  END_IF	
	END_IF
	
		IF arrAxisCtrl[AxiseNo.AxisName.AnDTCarryingUpDown].Cmd.arrbRealPoint[4] AND
           (( arrAxisCtrl[AxiseNo.AxisName.AnCarryingUpDown].Cmd.arrbRealPoint[4] AND  arrAxisCtrl[AxiseNo.AxisName.CaDTCarryingUpDown].Cmd.arrbRealPoint[4] )OR NOT Ca_OverNGMark)  THEN
			  DP_Step5:=6666;	
		END_IF

END_CASE


(**********************负极OH闭环纠偏************************************)
	//负极对齐度闭环计算  20240415SJ
 IF  Mach_Control.Ca_b.Ca_Quantited =0 THEN
		   iCaOverhandCount1_Y:=1; 
		   fCaSUMMean_Y:=0;
		   iCaOverhandCount2_Y:=0;   
END_IF
 IF  Mach_Control.Ca_b.Ca_Quantited =0 THEN
		   iCaOverhandCount1_X:=1; 
		   fCaSUMMean_X:=0;
		   iCaOverhandCount2_X:=0;   
END_IF


CASE DP_Step6 OF
101:
    IF Ca_OverNGMark THEN
        DP_Step6:=6666;
	ELSIF (CCD.Over.Finish.OverhandResult=4 OR CCD.Over.Finish.OverhandResult=2 OR CCD.Over.Finish.OverhandResult=1 ) AND NOT Ca_Number 
		AND( (arrAxisCtrl[AxiseNo.VirAxisName.VirMain].Status.fActPos>10 AND  arrAxisCtrl[AxiseNo.VirAxisName.VirMain].Status.fActPos<235) (*OR (arrAxisCtrl[AxiseNo.VirAxisName.VirMain].Status.fActPos=360)*)) THEN		
		DP_Step6:=102;
	ELSIF Ca_Number OR Mach_Control.U.EmptyRunMode OR Mach_Control.DT_b.DT_Overhang THEN//负极报警，空跑模式，Overhang屏蔽直接跳过
		DP_Step6:=6666;
	ELSIF NOT Ca_Number AND arrAxisCtrl[AxiseNo.VirAxisName.VirMain].Status.fActPos>235 AND arrAxisCtrl[AxiseNo.VirAxisName.VirMain].Status.fActPos<360 
		AND  CCD.Over.Finish.OverhandResult=0   THEN
		Mach_Control.Ca_b.Error[25]:=TRUE;//负极极片对齐度检测返回结果超时
		Par.stDT_date.Overhang_CSJS:=Par.stDT_date.Overhang_CSJS+1;
		DP_Step6:=6666;
	ELSIF CCD.Over.Finish.OverhandResult=3   THEN		
		Mach_Control.Ca_b.Error[27]:=TRUE;  //负极极片对齐度检测返回结果无片报警
		DP_Step6:=102;
	END_IF
					
102:
	CellMemory[Mach_Control.DT_b.DT_Memory].Overhang_Result[CCD.Over.Start.iPliesNo]:=CCD.Over.Finish.OverhandResult;	
	CellMemory[Mach_Control.DT_b.DT_Memory].DiaphragmUnwindingTension2[CCD.Over.Start.iPliesNo]:=LIMIT(150, Mach_Control.DT_b.DiaphragmUnwindingTension,250);
	CellMemory[Mach_Control.DT_b.DT_Memory].Ca_Ear_Overhang_A_C[Mach_Control.Ca_b.Ca_Quantited]:=ABS(CCD.Over.Finish.AnCaOverhandX1);
	CellMemory[Mach_Control.DT_b.DT_Memory].Ca_Ear_Overhang_S_CIL[Mach_Control.Ca_b.Ca_Quantited]:=ABS(CCD.Over.Finish.PoleOverhandX1);
	CellMemory[Mach_Control.DT_b.DT_Memory].Ca_Ear_No_Overhang_A_C[Mach_Control.Ca_b.Ca_Quantited]:=ABS(CCD.Over.Finish.AnCaOverhandX4);
	CellMemory[Mach_Control.DT_b.DT_Memory].Ca_Ear_No_Overhang_S_A[Mach_Control.Ca_b.Ca_Quantited]:=ABS(CCD.Over.Finish.PoleOverhandX4);
	
	CellMemory[Mach_Control.DT_b.DT_Memory].Ca_Ear_L_Overhang_A_C[Mach_Control.Ca_b.Ca_Quantited]:=ABS(CCD.Over.Finish.AnCaOverhandY1);
	CellMemory[Mach_Control.DT_b.DT_Memory].Ca_Ear_L_Overhang_S_A[Mach_Control.Ca_b.Ca_Quantited]:=ABS(CCD.Over.Finish.PoleOverhandY1);
	CellMemory[Mach_Control.DT_b.DT_Memory].Ca_Ear_R_Overhang_A_C[Mach_Control.Ca_b.Ca_Quantited]:=ABS(CCD.Over.Finish.AnCaOverhandY4);
	CellMemory[Mach_Control.DT_b.DT_Memory].Ca_Ear_R_Overhang_S_A[Mach_Control.Ca_b.Ca_Quantited]:=ABS(CCD.Over.Finish.PoleOverhandY4);
	
	CellMemory[Mach_Control.DT_b.DT_Memory].Ca_Cell_Overhang:=ABS(CCD.Over.Finish.AddOverhangX1);
	CellMemory[Mach_Control.DT_b.DT_Memory].Ca_Cell_Overhang_No:=ABS(CCD.Over.Finish.AddOverhangX4);
	CellMemory[Mach_Control.DT_b.DT_Memory].Ca_Cell_Overhang_L:=ABS(CCD.Over.Finish.AddOverhangY1);
	CellMemory[Mach_Control.DT_b.DT_Memory].Ca_Cell_Overhang_R:=ABS(CCD.Over.Finish.AddOverhangY4);
	
	CellMemory[Mach_Control.DT_b.DT_Memory].Ca_PoleOverhandX2[Mach_Control.Ca_b.Ca_Quantited]:=ABS(CCD.Over.Finish.PoleOverhandX2);
	CellMemory[Mach_Control.DT_b.DT_Memory].Ca_PoleOverhandX3[Mach_Control.Ca_b.Ca_Quantited]:=ABS(CCD.Over.Finish.PoleOverhandX3);
	CellMemory[Mach_Control.DT_b.DT_Memory].Ca_PoleOverhandY2[Mach_Control.Ca_b.Ca_Quantited]:=ABS(CCD.Over.Finish.PoleOverhandY2);
	CellMemory[Mach_Control.DT_b.DT_Memory].Ca_PoleOverhandY3[Mach_Control.Ca_b.Ca_Quantited]:=ABS(CCD.Over.Finish.PoleOverhandY3);
	
	CellMemory[Mach_Control.DT_b.DT_Memory].Ca_AnCaOverhandX2[Mach_Control.Ca_b.Ca_Quantited]:=ABS(CCD.Over.Finish.AnCaOverhandX2);
	CellMemory[Mach_Control.DT_b.DT_Memory].Ca_AnCaOverhandX3[Mach_Control.Ca_b.Ca_Quantited]:=ABS(CCD.Over.Finish.AnCaOverhandX3);
	CellMemory[Mach_Control.DT_b.DT_Memory].Ca_AnCaOverhandY2[Mach_Control.Ca_b.Ca_Quantited]:=ABS(CCD.Over.Finish.AnCaOverhandY2);
	CellMemory[Mach_Control.DT_b.DT_Memory].Ca_AnCaOverhandY3[Mach_Control.Ca_b.Ca_Quantited]:=ABS(CCD.Over.Finish.AnCaOverhandY3);
	
	CellMemory[Mach_Control.DT_b.DT_Memory].Ca_AddOverhangX2:=ABS(CCD.Over.Finish.AddOverhangX2);
	CellMemory[Mach_Control.DT_b.DT_Memory].Ca_AddOverhangX3:=ABS(CCD.Over.Finish.AddOverhangX3);
	CellMemory[Mach_Control.DT_b.DT_Memory].Ca_AddOverhangY2:=ABS(CCD.Over.Finish.AddOverhangY2);
	CellMemory[Mach_Control.DT_b.DT_Memory].Ca_AddOverhangY3:=ABS(CCD.Over.Finish.AddOverhangY3);
	
	CellMemory[Mach_Control.DT_b.DT_Memory].Ca_MQ_Slice[Mach_Control.Ca_b.Ca_Quantited]:=Par.stDT_date.Ca_MQ_Slice[9];
	
	CellMemory[Mach_Control.DT_b.DT_Memory].Chipdata[CCD.Over.Start.iPliesNo].Serialnumber:=CCD.Over.Start.iPliesNo;
	CellMemory[Mach_Control.DT_b.DT_Memory].Chipdata[CCD.Over.Start.iPliesNo].Polarity:=1;
	CellMemory[Mach_Control.DT_b.DT_Memory].Chipdata[CCD.Over.Start.iPliesNo].Platenumber:=Par.stDT_date.Ca_MQ_Slice[9].stPoleNo;
	CellMemory[Mach_Control.DT_b.DT_Memory].Chipdata[CCD.Over.Start.iPliesNo].CalapTen:=Par.stDT_date.Ca_MQ_Slice[9].UnreelingTension;
	CellMemory[Mach_Control.DT_b.DT_Memory].Chipdata[CCD.Over.Start.iPliesNo].GMlapTen:=LIMIT(150, Mach_Control.DT_b.DiaphragmUnwindingTension,250);
	CellMemory[Mach_Control.DT_b.DT_Memory].Chipdata[CCD.Over.Start.iPliesNo].GMlapRectify:=LIMIT( Par.stDT_date.fRectifyBalanceValue-0.2,  Mach_Control.DT_b.RecDevPV,Par.stDT_date.fRectifyBalanceValue+0.2);
	
	Ca_AlarmTON[11].IN:=FALSE;
	
	IF  CCD.Over.Finish.OverhandResult=1 THEN
		//计算当前 Y1 Y2    Y3 Y4中值
       fCaMeanSingle_Y:= ( (CCD.Over.Finish.AnCaOverhandY1+CCD.Over.Finish.AnCaOverhandY2)*0.5 - (CCD.Over.Finish.AnCaOverhandY3+CCD.Over.Finish.AnCaOverhandY4)*0.5 )*0.5;  //当前片Y方向 
	   fCaSUMMean_Y:=fCaSUMMean_Y+fCaMeanSingle_Y;
	   iCaOverhandCount2_Y:=iCaOverhandCount2_Y+1;

		//计算当前 X2 X4   X1 X3中值
       fCaMeanSingle_X:= (   ( (CCD.Over.Finish.AnCaOverhandX2+CCD.Over.Finish.AnCaOverhandX4)*0.5-1)   -  ( (CCD.Over.Finish.AnCaOverhandX1+CCD.Over.Finish.AnCaOverhandX3)*0.5-1.5 )   )*0.5;  //当前片Y方向 
	   fCaSUMMean_X:=fCaSUMMean_X+fCaMeanSingle_X;
	   iCaOverhandCount2_X:=iCaOverhandCount2_X+1;	
	END_IF   
			  //到达20层后计算一次Y
		IF  NOT   Mach_Control.DT_b.DT_OHclosure THEN	  
				IF  Mach_Control.Ca_b.Ca_Quantited>=iCaOverhandCount1_Y*10     THEN
					
						 IF  iCaOverhandCount2_Y>=3 THEN   
							fCaArvMean_Y:=fCaSUMMean_Y/iCaOverhandCount2_Y;
						ELSE
							fCaArvMean_Y:=0;
						 END_IF
						 fCaOffsetMean_Y:=LIMIT( -0.5,  fCaArvMean_Y*0.5 ,0.5  )  ;                    //SEL(fCaArvMean>0.1,  0 , fCaArvMean*0.333 )   ;
						 
						 iCaOverhandCount1_Y:=iCaOverhandCount1_Y+1;
						 fCaSUMMean_Y:=0;
						 iCaOverhandCount2_Y:=0;
				END_IF
				   
						  //到达20层后计算一次X
				IF  Mach_Control.Ca_b.Ca_Quantited>=iCaOverhandCount1_X*10     THEN
					
						 IF  iCaOverhandCount2_X>=3 THEN   
							fCaArvMean_X:=fCaSUMMean_X/iCaOverhandCount2_X;
						ELSE
							fCaArvMean_X:=0;
						 END_IF
						 fCaOffsetMean_X:=LIMIT( -0.5,   fCaArvMean_X*0.5 ,0.5  )  ;                    //SEL(fCaArvMean>0.1,  0 , fCaArvMean*0.333 )   ;
						 
						 iCaOverhandCount1_X:=iCaOverhandCount1_X+1;
						 fCaSUMMean_X:=0;
						 iCaOverhandCount2_X:=0;
				END_IF
		ELSE		
				 fCaOffsetMean_Y:=0;
				 fCaOffsetMean_X:=0;
        END_IF 


	   
	DP_Step6:=103;	


103:
	//CCD.Over.Finish.OverhandResult:=0;
	DP_Step6:=6666;	


END_CASE







CASE DP_Step7 OF
201:
    IF An_OverNGMark THEN
       DP_Step7:=6666;	
	ELSIF (CCD.Over.Finish.OverhandResult=4 OR CCD.Over.Finish.OverhandResult=2 OR CCD.Over.Finish.OverhandResult=1 ) AND NOT An_Number 
		AND ((arrAxisCtrl[AxiseNo.VirAxisName.VirMain].Status.fActPos>10 AND  arrAxisCtrl[AxiseNo.VirAxisName.VirMain].Status.fActPos<235)(* OR
		 (arrAxisCtrl[AxiseNo.VirAxisName.VirMain].Status.fActPos=360)*))THEN
		DP_Step7:=202;
	ELSIF An_Number OR Mach_Control.U.EmptyRunMode OR Mach_Control.DT_b.DT_Overhang THEN//负极报警，空跑模式，Overhang屏蔽直接跳过
		DP_Step7:=6666;	
	ELSIF   NOT An_Number AND arrAxisCtrl[AxiseNo.VirAxisName.VirMain].Status.fActPos>235 AND arrAxisCtrl[AxiseNo.VirAxisName.VirMain].Status.fActPos<360 
		AND CCD.Over.Finish.OverhandResult=0 THEN
		Mach_Control.An_b.Error[25]:=TRUE;//正极极片对齐度检测返回结果超时
		Par.stDT_date.Overhang_CSJS:=Par.stDT_date.Overhang_CSJS+1;
		DP_Step7:=6666;	
	ELSIF CCD.Over.Finish.OverhandResult=3 THEN 		
		Mach_Control.An_b.Error[27]:=TRUE; //正极极片对齐度检测返回结果无片报警
		DP_Step7:=202;	
	END_IF
							
											
202:
	CellMemory[Mach_Control.DT_b.DT_Memory].Overhang_Result[CCD.Over.Start.iPliesNo]:=CCD.Over.Finish.OverhandResult;	
	CellMemory[Mach_Control.DT_b.DT_Memory].DiaphragmUnwindingTension2[CCD.Over.Start.iPliesNo]:=LIMIT(150, Mach_Control.DT_b.DiaphragmUnwindingTension,250);
	CellMemory[Mach_Control.DT_b.DT_Memory].An_Ear_Overhang_A_C[Mach_Control.An_b.An_Quantited]:=ABS(CCD.Over.Finish.AnCaOverhandX1);
	CellMemory[Mach_Control.DT_b.DT_Memory].An_Ear_Overhang_S_CIL[Mach_Control.An_b.An_Quantited]:=ABS(CCD.Over.Finish.PoleOverhandX1);
	CellMemory[Mach_Control.DT_b.DT_Memory].An_Ear_No_Overhang_A_C[Mach_Control.An_b.An_Quantited]:=ABS(CCD.Over.Finish.AnCaOverhandX4);
	CellMemory[Mach_Control.DT_b.DT_Memory].An_Ear_No_Overhang_S_A[Mach_Control.An_b.An_Quantited]:=ABS(CCD.Over.Finish.PoleOverhandX4);
	
	CellMemory[Mach_Control.DT_b.DT_Memory].An_Ear_L_Overhang_A_C[Mach_Control.An_b.An_Quantited]:=ABS(CCD.Over.Finish.AnCaOverhandY1);
	CellMemory[Mach_Control.DT_b.DT_Memory].An_Ear_L_Overhang_S_A[Mach_Control.An_b.An_Quantited]:=ABS(CCD.Over.Finish.PoleOverhandY1);
	CellMemory[Mach_Control.DT_b.DT_Memory].An_Ear_R_Overhang_A_C[Mach_Control.An_b.An_Quantited]:=ABS(CCD.Over.Finish.AnCaOverhandY4);
	CellMemory[Mach_Control.DT_b.DT_Memory].An_Ear_R_Overhang_S_A[Mach_Control.An_b.An_Quantited]:=ABS(CCD.Over.Finish.PoleOverhandY4);
	
	CellMemory[Mach_Control.DT_b.DT_Memory].An_Cell_Overhang:=ABS(CCD.Over.Finish.AddOverhangX1);
	CellMemory[Mach_Control.DT_b.DT_Memory].An_Cell_Overhang_No:=ABS(CCD.Over.Finish.AddOverhangX4);
	CellMemory[Mach_Control.DT_b.DT_Memory].An_Cell_Overhang_L:=ABS(CCD.Over.Finish.AddOverhangY1);
	CellMemory[Mach_Control.DT_b.DT_Memory].An_Cell_Overhang_R:=ABS(CCD.Over.Finish.AddOverhangY4);
	
	CellMemory[Mach_Control.DT_b.DT_Memory].An_PoleOverhandX2[Mach_Control.An_b.An_Quantited]:=ABS(CCD.Over.Finish.PoleOverhandX2);
	CellMemory[Mach_Control.DT_b.DT_Memory].An_PoleOverhandX3[Mach_Control.An_b.An_Quantited]:=ABS(CCD.Over.Finish.PoleOverhandX3);
	CellMemory[Mach_Control.DT_b.DT_Memory].An_PoleOverhandY2[Mach_Control.An_b.An_Quantited]:=ABS(CCD.Over.Finish.PoleOverhandY2);
	CellMemory[Mach_Control.DT_b.DT_Memory].An_PoleOverhandY3[Mach_Control.An_b.An_Quantited]:=ABS(CCD.Over.Finish.PoleOverhandY3);
	
	CellMemory[Mach_Control.DT_b.DT_Memory].An_AnCaOverhandX2[Mach_Control.An_b.An_Quantited]:=ABS(CCD.Over.Finish.AnCaOverhandX2);
	CellMemory[Mach_Control.DT_b.DT_Memory].An_AnCaOverhandX3[Mach_Control.An_b.An_Quantited]:=ABS(CCD.Over.Finish.AnCaOverhandX3);
	CellMemory[Mach_Control.DT_b.DT_Memory].An_AnCaOverhandY2[Mach_Control.An_b.An_Quantited]:=ABS(CCD.Over.Finish.AnCaOverhandY2);
	CellMemory[Mach_Control.DT_b.DT_Memory].An_AnCaOverhandY3[Mach_Control.An_b.An_Quantited]:=ABS(CCD.Over.Finish.AnCaOverhandY3);
	
	CellMemory[Mach_Control.DT_b.DT_Memory].An_AddOverhangX2:=ABS(CCD.Over.Finish.AddOverhangX2);
	CellMemory[Mach_Control.DT_b.DT_Memory].An_AddOverhangX3:=ABS(CCD.Over.Finish.AddOverhangX3);
	CellMemory[Mach_Control.DT_b.DT_Memory].An_AddOverhangY2:=ABS(CCD.Over.Finish.AddOverhangY2);
	CellMemory[Mach_Control.DT_b.DT_Memory].An_AddOverhangY3:=ABS(CCD.Over.Finish.AddOverhangY3);
	
	CellMemory[Mach_Control.DT_b.DT_Memory].An_MQ_Slice[Mach_Control.An_b.An_Quantited]:=Par.stDT_date.An_MQ_Slice[2];
	
	CellMemory[Mach_Control.DT_b.DT_Memory].Chipdata[CCD.Over.Start.iPliesNo].Serialnumber:=CCD.Over.Start.iPliesNo;
	CellMemory[Mach_Control.DT_b.DT_Memory].Chipdata[CCD.Over.Start.iPliesNo].Polarity:=2;
	CellMemory[Mach_Control.DT_b.DT_Memory].Chipdata[CCD.Over.Start.iPliesNo].Platenumber:=Par.stDT_date.An_MQ_Slice[2].stPoleNo;
	CellMemory[Mach_Control.DT_b.DT_Memory].Chipdata[CCD.Over.Start.iPliesNo].AnlapTen:=Par.stDT_date.An_MQ_Slice[2].UnreelingTension;
	CellMemory[Mach_Control.DT_b.DT_Memory].Chipdata[CCD.Over.Start.iPliesNo].GMlapTen:=LIMIT(150, Mach_Control.DT_b.DiaphragmUnwindingTension,250);
	CellMemory[Mach_Control.DT_b.DT_Memory].Chipdata[CCD.Over.Start.iPliesNo].GMlapRectify:=LIMIT( Par.stDT_date.fRectifyBalanceValue-0.2,  Mach_Control.DT_b.RecDevPV,Par.stDT_date.fRectifyBalanceValue+0.2);

	
	DP_Step7:=203;	

203:
	//CCD.Over.Finish.OverhandResult:=0;
	DP_Step7:=6666;

END_CASE



CASE DP_Step8 OF	
100:
	Ca_StandbySub3_ton[2].IN:=FALSE;
	IF  NOT Mach_Control.U.CCD_ChosesHMI  AND NOT  Mach_Control.U.EmptyRunMode (*AND NOT An_OverhangNG*) THEN
		//IF arrAxis[AxiseNo.VirAxisName.VirMain].NcToPlc.SetPos>109 AND arrAxis[AxiseNo.VirAxisName.VirMain].NcToPlc.SetPos<=112   THEN
		IF arrAxis[AxiseNo.VirAxisName.VirMain].NcToPlc.SetPos>122.5 AND arrAxis[AxiseNo.VirAxisName.VirMain].NcToPlc.SetPos<=128   THEN
				CCD.CaRec.Finish.RectifyX1:=0;
				CCD.CaRec.Finish.RectifyX2:=0;
				CCD.CaRec.Finish.RectifyY:=0;		
				CCD.CaRec.Finish.RectifyResult:=0;//拍照结果清零									
				Mach_Control.Ca_b.Ca_CCDStart :=TRUE;//启动CCD拍照
				CCD.CaRec.Start.iPhotoDo:=1;//启动CCD第二次拍照
				//arrCyCtrl[arrCyNo.ElectValveName.CadeviationIonizedWind].Cmd.bON:=TRUE;//负极纠偏平台除尘
				//arrCyCtrl[arrCyNo.ElectValveName.AndeviationIonizedWind].Cmd.bON:=TRUE;//正极纠偏平台除尘
				DP_Step8:=110;
		END_IF
	ELSE
		DP_Step8:=6661;
	END_IF
110:
	Ca_StandbySub3_ton[2].IN:=CCD.CaRec.Finish.RectifyResult=0;
	IF Ca_StandbySub3_ton[2].Q THEN
		Mach_Control.DT_b.Error[51]:=TRUE;//检测负极纠偏平台空片结果返回超时
		DP_Step8:=9991;
	ELSIF CCD.CaRec.Finish.RectifyResult<>0 AND CCD.CaRec.Finish.RectifyResult<>3   THEN
		Mach_Control.Ca_b.Error[24]:=TRUE;//负极纠偏平台NG片未排掉报警，请拿掉
		Ca_StandbySub3_ton[2].IN:=FALSE;
		DP_Step8:=9992;
	ELSIF CCD.CaRec.Finish.RectifyResult=3  THEN
		DP_Step8:=6661;
	END_IF

200:
	An_StandbySub3_ton[2].IN:=FALSE;
	IF  NOT Mach_Control.U.CCD_ChosesHMI  AND NOT  Mach_Control.U.EmptyRunMode  (*AND NOT Ca_OverhangNG*) THEN
		//IF arrAxis[AxiseNo.VirAxisName.VirMain].NcToPlc.SetPos>118 AND arrAxis[AxiseNo.VirAxisName.VirMain].NcToPlc.SetPos<=123  THEN
		IF arrAxis[AxiseNo.VirAxisName.VirMain].NcToPlc.SetPos>122.5 AND arrAxis[AxiseNo.VirAxisName.VirMain].NcToPlc.SetPos<=128   THEN
			CCD.AnRec.Finish.RectifyResult:=0;
			CCD.AnRec.Finish.RectifyX1:=0;
			CCD.AnRec.Finish.RectifyX2:=0;
			CCD.AnRec.Finish.RectifyY:=0;												
			Mach_Control.An_b.An_CCDStart :=TRUE;//启动CCD拍照
			CCD.AnRec.Start.iPhotoDo:=1;//第二次拍照
			//arrCyCtrl[arrCyNo.ElectValveName.CadeviationIonizedWind].Cmd.bON:=TRUE;//负极纠偏平台除尘
			//arrCyCtrl[arrCyNo.ElectValveName.AndeviationIonizedWind].Cmd.bON:=TRUE;//正极纠偏平台除尘
			DP_Step8:=210;
		END_IF
	ELSE
		DP_Step8:=6662;
	END_IF	
210:
	An_StandbySub3_ton[2].IN:=CCD.AnRec.Finish.RectifyResult=0;
	IF An_StandbySub3_ton[2].Q THEN				
		Mach_Control.DT_b.Error[52]:=TRUE;//检测正极纠偏平台空片结果返回超时
		An_StandbySub3_ton[2].IN:=FALSE;
		DP_Step8:=9993;		
	ELSIF CCD.AnRec.Finish.RectifyResult<>0 AND CCD.AnRec.Finish.RectifyResult<>3 THEN
		Mach_Control.An_b.Error[24]:=TRUE;//正极纠偏平台NG片未排掉报警，请拿掉 
		An_StandbySub3_ton[2].IN:=FALSE;
		DP_Step8:=9994;
	ELSIF CCD.AnRec.Finish.RectifyResult=3 THEN
		An_StandbySub3_ton[2].IN:=FALSE;
		DP_Step8:=6662;
	END_IF
	
END_CASE





(*
////////////////////////////////////////////////////////////////////////////////////运行中处理 流程//////////////////////////////////////////////////////////////////////////////////////////////
//主轴在运行时，真空、破真空，以及是否能取片、有无料标记
(*
IF VirMain_TagatTime<1 THEN
		CamOutArgel:=0.47*VirMain_TagatTime*360;
ELSE
		CamOutArgel:=160;
END_IF
*)

CamOutArgel:=170;

CASE DP_Step3 OF 
100://负极叠片，正极在取片位
	bStandbyStep1_1:=FALSE;
	bStandbyStep1_2:=FALSE;
	DP_Step3:=110; 
110:   //叠负极片同时 判断证据能否取片  提高效率
	IF arrAxisCtrl[AxiseNo.VirAxisName.VirMain].Status.fActPos>=10  AND  arrAxisCtrl[AxiseNo.VirAxisName.VirMain].Status.fActPos<=220     THEN
	//正送片搬运极取片处理
		IF   arrAxisCtrl[AxiseNo.AxisName.AnCarryingUpDown].Cmd.arrbRealPoint[4] AND 
			  NOT Mach_Control.An_b.An_CarryingFalg    AND  ( Mach_Control.An_b.An_MainBeltOK OR  Mach_Control.U.EmptyRunMode )  AND 
			  NOT  Mach_Control.An_b.An_MainBelting   AND NOT  bStandbyStep1_1 AND (NOT An_JumpRules[3]  AND NOT  An_JumpRules[6] AND NOT An_JumpRules[8] AND NOT An_JumpRules[10])(*AND NOT Mach_Control.An_b.JumpPiceReady *) THEN
			   An_Step0:=10;//正极取流水线子程序
			   bStandbyStep1_1:=TRUE;
		END_IF
		
		IF arrAxisCtrl[AxiseNo.AxisName.AnDTCarryingUpDown].Cmd.arrbRealPoint[4] AND 
		 Mach_Control.An_b.An_deviationDPOK AND NOT Mach_Control.An_b.An_DPCarryingFalg AND  
			Mach_Control.An_b.An_deviationFalg  AND  NOT  bStandbyStep1_2  AND NOT DP_CheseCam  THEN
			An_Step3:=10;//正极取纠偏平台子程序
			bStandbyStep1_2:=TRUE;
		END_IF
	
	ELSIF  arrAxisCtrl[AxiseNo.VirAxisName.VirMain].Status.fActPos>220  THEN
		DP_Step3:=120;
	END_IF		   
	
	
120:
	arrCyCtrl[arrCyNo.ElectValveName.CadeviationVacuum].Cmd.bON:=TRUE;//负极纠偏平台真空开			
	arrCyCtrl[arrCyNo.ElectValveName.CadeviationVacuum].Cmd.bOFF:=FALSE;//负极纠偏平台真空开					
	IF 	arrAxisCtrl[AxiseNo.VirAxisName.VirMain].Status.fActPos>=234 THEN//198
		
		Mach_Control.Ca_b.Ca_Rectifydev_CS:=0;
		CCD.Over.Start.stPoleNo:=Par.stDT_date.Ca_MQ_Slice[8].stPoleNo;
		arrCyCtrl[arrCyNo.ElectValveName.CaDTCarryingVacuum].Cmd.bON:=TRUE;//负极叠片搬运真空破
		arrCyCtrl[arrCyNo.ElectValveName.CaDTCarryingVacuum].Cmd.bOFF:=FALSE;//负极叠片搬运真空破
		arrCyCtrl[arrCyNo.ElectValveName.CaCarryingVacuum2].Cmd.bON:=TRUE;//负极送片搬运真空破
		arrCyCtrl[arrCyNo.ElectValveName.CaCarryingVacuum2].Cmd.bOFF:=FALSE;//负极送片搬运真空破
		arrCyCtrl[arrCyNo.ElectValveName.CadeviationVacuum].Cmd.bON:=TRUE;//负极纠偏平台真空开
		arrCyCtrl[arrCyNo.ElectValveName.CadeviationVacuum].Cmd.bOFF:=FALSE;//负极纠偏平台真空开			
		
		Mach_Control.Ca_b.Ca_DPCarryingFalg :=FALSE;//复位负极叠片搬运吸盘上有料标记
		//IF Mach_Control.Ca_b.Ca_CarryingFalg THEN
			Mach_Control.Ca_b.Ca_deviationFalg:=TRUE;//置位纠偏平台上有料标记
			Mach_Control.Ca_b.Ca_CarryingFalg:=FALSE;//复位负极送片搬运吸盘上有料标记
		//END_IF
		Par.stDT_date.Ca_MQ_Slice[8]:=Par.stDT_date.Ca_MQ_Slice[7];
		
	END_IF	
	IF 	arrAxisCtrl[AxiseNo.VirAxisName.VirMain].Status.fActPos>=342 THEN//198
     	CCD.Over.Start.iPliesNo:=UINT_TO_INT(Mach_Control.Ca_b.Ca_Quantited + Mach_Control.An_b.An_Quantited+1);	
		IF NOT Ca_Number THEN
			CCD.Over.Start.iPhotoDo:=1;
		ELSE
			CCD.Over.Start.iPhotoDo:=2;
		END_IF
		Mach_Control.DT_b.CDD_OverStart:=TRUE;
		DP_Step3:=121;
	 END_IF		
		
121:
	IF 	arrAxisCtrl[AxiseNo.VirAxisName.VirMain].Status.fActPos>=360 THEN//198
		arrCyCtrl[arrCyNo.ElectValveName.CaCarryingVacuum2].Cmd.bON:=FALSE;//负极送片搬运真空开
		arrCyCtrl[arrCyNo.ElectValveName.CaCarryingVacuum2].Cmd.bOFF:=TRUE;//负极送片搬运真空开
		arrCyCtrl[arrCyNo.ElectValveName.CaDTCarryingVacuum].Cmd.bON:=FALSE;//负极叠片搬运真空破
		arrCyCtrl[arrCyNo.ElectValveName.CaDTCarryingVacuum].Cmd.bOFF:=TRUE;//负极叠片搬运真空破
		DP_Step3:=6666;
	END_IF	
	
	
200://负极叠片，正极在取片位

	IF iAnCamInSel2=1 THEN
		arrCyCtrl[arrCyNo.ElectValveName.AnDTCarryingVacuum].Cmd.bON:=TRUE;//正极送片搬运真空关
		arrCyCtrl[arrCyNo.ElectValveName.AnDTCarryingVacuum].Cmd.bOFF:=FALSE;//正极送片搬运真空关
	END_IF
	
	//fbAnDTCarryingVacuum.Vacuumsel:=SEL(iAnCamInSel2=1,0,1)     ;//	正极叠片搬运真空开	
	IF arrAxisCtrl[AxiseNo.VirAxisName.VirMain].Status.fActPos>=210 THEN//复检提前
		IF Mach_Control.DT_b.DT_CCD_TwoModel THEN												
			CCD.AnRec.Finish.RectifyResult:=0;
			CCD.AnRec.Finish.RectifyX1:=0;
			CCD.AnRec.Finish.RectifyX2:=0;
			CCD.AnRec.Finish.RectifyY:=0;												
			Mach_Control.An_b.An_CCDStart :=TRUE;//启动CCD拍照
			CCD.AnRec.Start.iPhotoDo:=2;//第二次拍照	
		END_IF
		DP_Step3:=205;
	END_IF
205:			
	IF NOT DP_CheseCam  AND NOT  An_JumpRules[3]  AND NOT  An_JumpRules[6] AND NOT An_JumpRules[8] AND NOT An_JumpRules[10] THEN
	
		IF arrAxisCtrl[AxiseNo.VirAxisName.VirMain].Status.fActPos>=225  AND arrAxisCtrl[AxiseNo.VirAxisName.VirMain].Status.fActPos<=230 THEN	
			//fbAnCamInCarryingUpDown.bCamInExecute:=FALSE;//正极升解除耦合															
			//fbAnCamInCarryingWhirling.bCamInExecute:=FALSE;//正极旋转解除耦合			
			//Mach_Control.An_b.An_MainBelting:=FALSE;//正极搬运升降取极片中																					
			IF  NOT  Mach_Control.Ca_b.Ca_deviationFPOK  THEN    //负极放片纠偏太未在初始位置报警  
					Mach_Control.Ca_b.Error_tips[1]:=TRUE ;
			END_IF											
			IF  NOT  Mach_Control.An_b.An_deviationDPOK  THEN    //正极取片纠偏未完成报警
					Mach_Control.An_b.Error_tips[1]:=TRUE;
			END_IF			
			IF Mach_Control.An_b.An_deviationDPOK OR Mach_Control.U.EmptyRunMode OR	TRUE  THEN // 
				arrCyCtrl[arrCyNo.ElectValveName.AnDTCarryingVacuum].Cmd.bON:=TRUE;//正极叠片搬运真空开	
				arrCyCtrl[arrCyNo.ElectValveName.AnDTCarryingVacuum].Cmd.bOFF:=FALSE;//正极叠片搬运真空开		
				An_deviationDPOKFalg:=TRUE;	
			ELSE		
				arrCyCtrl[arrCyNo.ElectValveName.AnDTCarryingVacuum].Cmd.bON:=FALSE;//正极叠片搬运真空开					
				arrCyCtrl[arrCyNo.ElectValveName.AnDTCarryingVacuum].Cmd.bOFF:=TRUE;//正极叠片搬运真空开												
				fbAnCamInDTCarryingUpDown.bCamInExecute:=FALSE;	//正极叠片搬运升降凸轮解耦				
				IF NOT arrAxisCtrl[AxiseNo.AxisName.AnDTCarryingUpDown].Cmd.arrbRealPoint[4]    THEN
						arrAxisCtrl[AxiseNo.AxisName.AnDTCarryingUpDown].Cmd.iGoSetPos:=4;   //到等待位
				END_IF			
			END_IF	
			//IF NOT Mach_Control.An_b.JumpPiceReady THEN
				An_Step0:=10;//调用正极取片程序	
			//END_IF
			DP_Step3:=210;														
		END_IF									
	ELSE
			DP_Step3:=210;	
	END_IF


210:
	//打开或关闭真空，标记对应位置有料
	IF 	arrAxisCtrl[AxiseNo.VirAxisName.VirMain].Status.fActPos>=234 THEN//198
	
		Mach_Control.Ca_b.Ca_Rectifydev_CS:=0;
		arrCyCtrl[arrCyNo.ElectValveName.CaCarryingVacuum2].Cmd.bON:=TRUE;//负极送片搬运真空关
		arrCyCtrl[arrCyNo.ElectValveName.CaCarryingVacuum2].Cmd.bOFF:=FALSE;//负极送片搬运真空关
		arrCyCtrl[arrCyNo.ElectValveName.CaDTCarryingVacuum].Cmd.bON:=TRUE;//负极叠片搬运直空关
		arrCyCtrl[arrCyNo.ElectValveName.CaDTCarryingVacuum].Cmd.bOFF:=FALSE;//负极叠片搬运直空关
		arrCyCtrl[arrCyNo.ElectValveName.CadeviationVacuum].Cmd.bON:=TRUE;//负极纠偏平台真空开	
		arrCyCtrl[arrCyNo.ElectValveName.CadeviationVacuum].Cmd.bOFF:=FALSE;//负极纠偏平台真空开		
		
		Mach_Control.Ca_b.Ca_DPCarryingFalg :=FALSE;//复位负极叠片搬运吸盘上有料标记
		//IF Mach_Control.Ca_b.Ca_CarryingFalg THEN
			Mach_Control.Ca_b.Ca_deviationFalg:=TRUE;//置位纠偏平台上有料标记
			Mach_Control.Ca_b.Ca_CarryingFalg:=FALSE;//复位负极送片搬运吸盘上有料标记
		//END_IF
		Par.stDT_date.Ca_MQ_Slice[8]:=Par.stDT_date.Ca_MQ_Slice[7];
		IF An_deviationDPOKFalg AND  iAnCamInSel2=1   THEN
			Par.stDT_date.An_MQ_Slice[2]:=Par.stDT_date.An_MQ_Slice[1];
			//IF Mach_Control.An_b.An_deviationFalg THEN
				Mach_Control.An_b.An_DPCarryingFalg :=TRUE;//复位正极叠片搬运吸盘上有料标记										
				Mach_Control.An_b.An_deviationFalg:=FALSE;//置位纠偏平台上有料标记	
			//END_IF										
			arrCyCtrl[arrCyNo.ElectValveName.AndeviationVacuum].Cmd.bOFF:=TRUE;//正极纠偏平台真空关
			arrCyCtrl[arrCyNo.ElectValveName.AndeviationVacuum].Cmd.bON:=FALSE;//正极纠偏平台真空关
			arrCyCtrl[arrCyNo.ElectValveName.AndeviationVacuumBark].Cmd.bON:=TRUE;//正极纠偏平台破真空开	
			arrCyCtrl[arrCyNo.ElectValveName.AndeviationVacuumBark].Cmd.bOFF:=FALSE;//正极纠偏平台破真空开	
	(*	
		ELSIF NOT   DP_CheseCam THEN								
			An_Step3:=10;//正极叠片搬运取纠偏台极片	
	*)																					
		END_IF
	
	END_IF

	IF 	arrAxisCtrl[AxiseNo.VirAxisName.VirMain].Status.fActPos>=342 THEN//198
		CCD.Over.Start.iPliesNo:=UINT_TO_INT(Mach_Control.Ca_b.Ca_Quantited + Mach_Control.An_b.An_Quantited+1);
		CCD.Over.Start.stPoleNo:=Par.stDT_date.Ca_MQ_Slice[8].stPoleNo;
		IF NOT Ca_Number THEN
			CCD.Over.Start.iPhotoDo:=1;
		ELSE
			CCD.Over.Start.iPhotoDo:=2;
		END_IF
		Mach_Control.DT_b.CDD_OverStart:=TRUE;	
		IF NOT Ca_Number THEN
			DP_Step3:=211;					
		END_IF	
    END_IF	
211:
	IF 	arrAxisCtrl[AxiseNo.VirAxisName.VirMain].Status.fActPos>=360 THEN//198	
		arrCyCtrl[arrCyNo.ElectValveName.CaCarryingVacuum2].Cmd.bON:=FALSE;//负极送片搬运真空开
		arrCyCtrl[arrCyNo.ElectValveName.CaCarryingVacuum2].Cmd.bOFF:=TRUE;//负极送片搬运真空开
		arrCyCtrl[arrCyNo.ElectValveName.CaDTCarryingVacuum].Cmd.bON:=FALSE;//负极叠片搬运直空开
		arrCyCtrl[arrCyNo.ElectValveName.CaDTCarryingVacuum].Cmd.bOFF:=TRUE;//负极叠片搬运直空开
		DP_Step3:=6666;					
	END_IF
			



		
300://正极叠片，负极在取片位			
	bStandbyStep1_3:=FALSE;
	bStandbyStep1_4:=FALSE;
	DP_Step3:=310; 		
310:	
	IF arrAxisCtrl[AxiseNo.VirAxisName.VirMain].Status.fActPos>=10  AND  arrAxisCtrl[AxiseNo.VirAxisName.VirMain].Status.fActPos<=220     THEN
		//正送片搬运极取片处理
		IF   arrAxisCtrl[AxiseNo.AxisName.CaCarryingUpDown2].Cmd.arrbRealPoint[4] AND 
			NOT Mach_Control.Ca_b.Ca_CarryingFalg    AND  ( Mach_Control.Ca_b.Ca_CacheBeltDLOK OR  Mach_Control.U.EmptyRunMode )  AND 
			NOT  Mach_Control.Ca_b.Ca_CacheBelting   AND NOT  bStandbyStep1_3 THEN
			Ca_Step0:=10;   //负极取流水线子程序
			bStandbyStep1_3:=TRUE;
		END_IF
	
		IF arrAxisCtrl[AxiseNo.AxisName.CaDTCarryingUpDown].Cmd.arrbRealPoint[4] AND 
			Mach_Control.Ca_b.Ca_deviationDPOK AND NOT Mach_Control.Ca_b.Ca_DPCarryingFalg AND  
			Mach_Control.Ca_b.Ca_deviationFalg AND  NOT  bStandbyStep1_4   THEN
			Ca_Step3:=10;     //负极取纠偏平台子程序
			bStandbyStep1_4:=TRUE;
		END_IF					
	ELSIF  arrAxisCtrl[AxiseNo.VirAxisName.VirMain].Status.fActPos>220  THEN
			DP_Step3:=320; 
	END_IF	
	
320://正极叠片，负极在取片位
	arrCyCtrl[arrCyNo.ElectValveName.AndeviationVacuum].Cmd.bON:=TRUE;//正极纠偏平台真空开			
	arrCyCtrl[arrCyNo.ElectValveName.AndeviationVacuum].Cmd.bOFF:=FALSE;//正极纠偏平台真空开					
	IF 	arrAxisCtrl[AxiseNo.VirAxisName.VirMain].Status.fActPos>=234 THEN//198
	
		Mach_Control.An_b.An_Rectifydev_CS:=0;	
		arrCyCtrl[arrCyNo.ElectValveName.AnCarryingVacuum].Cmd.bON:=FALSE;//正极送片搬运真空关
		arrCyCtrl[arrCyNo.ElectValveName.AnCarryingVacuum].Cmd.bOFF:=TRUE;//正极送片搬运真空关
		arrCyCtrl[arrCyNo.ElectValveName.AnCarryingVacuumBark].Cmd.bON:=TRUE;//正极送片搬运破真空开
		arrCyCtrl[arrCyNo.ElectValveName.AnCarryingVacuumBark].Cmd.bOFF:=FALSE;//正极送片搬运破真空开
		
		arrCyCtrl[arrCyNo.ElectValveName.AnDTCarryingVacuum].Cmd.bON:=FALSE;//正极送片搬运真空关
		arrCyCtrl[arrCyNo.ElectValveName.AnDTCarryingVacuum].Cmd.bOFF:=TRUE;//正极送片搬运真空关
		arrCyCtrl[arrCyNo.ElectValveName.AnDTCarryingVacuumBark].Cmd.bON:=TRUE;//正极送片搬运破真空开
		arrCyCtrl[arrCyNo.ElectValveName.AnDTCarryingVacuumBark].Cmd.bOFF:=FALSE;//正极送片搬运破真空开
		
		arrCyCtrl[arrCyNo.ElectValveName.AndeviationVacuum].Cmd.bON:=TRUE;//正极纠偏平台真空开		
		arrCyCtrl[arrCyNo.ElectValveName.AndeviationVacuum].Cmd.bOFF:=FALSE;//正极纠偏平台真空开		
		
		
		Mach_Control.An_b.An_DPCarryingFalg :=FALSE;//复位正极叠片搬运吸盘上有料标记
		//IF Mach_Control.An_b.An_CarryingFalg THEN
			Mach_Control.An_b.An_deviationFalg:=TRUE;//置位纠偏平台上有料标记
			Mach_Control.An_b.An_CarryingFalg:=FALSE;//复位正极送片搬运吸盘上有料标记
		//END_IF
		Par.stDT_date.An_MQ_Slice[1]:=Par.stDT_date.An_MQ_Slice[0];
		
	END_IF
	
	IF 	arrAxisCtrl[AxiseNo.VirAxisName.VirMain].Status.fActPos>=342 THEN//198
		CCD.Over.Start.iPliesNo:=UINT_TO_INT(Mach_Control.Ca_b.Ca_Quantited + Mach_Control.An_b.An_Quantited+1);
		CCD.Over.Start.stPoleNo:=Par.stDT_date.An_MQ_Slice[2].stPoleNo;
		IF NOT An_Number THEN
			CCD.Over.Start.iPhotoDo:=1;
		ELSE
			CCD.Over.Start.iPhotoDo:=2;
		END_IF
		Mach_Control.DT_b.CDD_OverStart:=TRUE;				
		DP_Step3:=6666;	
	END_IF
400:	//复检提前------//正极叠片，负极在叠片位

	//fbCaDTCarryingVacuum.Vacuumsel:= SEL(iCaCamInSel2=1 ,0,1)   ;//	负极叠片搬运真空开
	IF iCaCamInSel2=1 THEN
		arrCyCtrl[arrCyNo.ElectValveName.CaDTCarryingVacuum].Cmd.bON:=FALSE;//负极叠台搬运真空开	
		arrCyCtrl[arrCyNo.ElectValveName.CaDTCarryingVacuum].Cmd.bOFF:=TRUE;//负极叠台搬运真空开		
	END_IF

	IF 	arrAxisCtrl[AxiseNo.VirAxisName.VirMain].Status.fActPos>=210 THEN//198
		IF Mach_Control.DT_b.DT_CCD_TwoModel THEN
				CCD.CaRec.Finish.RectifyX1:=0;
				CCD.CaRec.Finish.RectifyX2:=0;
				CCD.CaRec.Finish.RectifyY:=0;		
				CCD.CaRec.Finish.RectifyResult:=0;//拍照结果清零									
				Mach_Control.Ca_b.Ca_CCDStart :=TRUE;//启动CCD拍照
				CCD.CaRec.Start.iPhotoDo:=2;//启动CCD第二次拍照									
		END_IF
		DP_Step3:=405;
	END_IF
405:		
	IF arrAxisCtrl[AxiseNo.VirAxisName.VirMain].Status.fActPos>=225  AND arrAxisCtrl[AxiseNo.VirAxisName.VirMain].Status.fActPos<=230 THEN																								
		IF  NOT  Mach_Control.An_b.An_deviationFPOK  THEN    //正极放片纠偏太未在初始位置报警  
			  Mach_Control.An_b.Error_tips[2]:=TRUE ;
		END_IF
		
		IF  NOT  Mach_Control.Ca_b.Ca_deviationDPOK  THEN    //负极取片纠偏未完成报警
			  Mach_Control.Ca_b.Error_tips[2]:=TRUE ;
		END_IF		

		//正极叠片时平移到位后判断正极纠偏台是否允许放片
		IF Mach_Control.An_b.An_deviationFPOK OR Mach_Control.U.EmptyRunMode  THEN 
				An_deviationFPOKFalg:=TRUE;//正极纠偏平台允许放片标记
		ELSE									
			fbAnCamInCarryingUpDown.bCamInExecute:=FALSE;	//正极送片搬运升降凸轮解耦				
			IF NOT arrAxisCtrl[AxiseNo.AxisName.AnCarryingUpDown].Cmd.arrbRealPoint[4]    THEN
				arrAxisCtrl[AxiseNo.AxisName.AnCarryingUpDown].Cmd.iGoSetPos:=4;
			END_IF;				
		END_IF					
		IF Mach_Control.Ca_b.Ca_deviationDPOK OR Mach_Control.U.EmptyRunMode OR TRUE  THEN //  
			Ca_deviationDPOKFalg:=TRUE;	
			arrCyCtrl[arrCyNo.ElectValveName.CaDTCarryingVacuum].Cmd.bON:=FALSE;//负极叠片搬运真空开	
			arrCyCtrl[arrCyNo.ElectValveName.CaDTCarryingVacuum].Cmd.bOFF:=TRUE;//负极叠片搬运真空开		
		ELSE	
			//arrCyCtrl[arrCyNo.ElectValveName.CaDTCarryingVacuum].Cmd.bON:=FALSE;//负极叠片搬运真空开									
			fbCaCamInDTCarryingUpDown.bCamInExecute:=FALSE;	//负极叠片搬运升降凸轮解耦				
			IF NOT arrAxisCtrl[AxiseNo.AxisName.CaDTCarryingUpDown].Cmd.arrbRealPoint[4]    THEN
				arrAxisCtrl[AxiseNo.AxisName.CaDTCarryingUpDown].Cmd.iGoSetPos:=4;   //到等待位
			ELSE
				arrAxisCtrl[AxiseNo.AxisName.CaDTCarryingUpDown].Cmd.iGoSetPos:=0;   //到等待位
			END_IF;				
		END_IF									
		Ca_Step0:=10;//调用负极取片程序       取片允许条件在子程序里
		DP_Step3:=410;		
	END_IF
(*	
	//判断是否允许负极送片搬运取料
	IF arrAxisCtrl[AxiseNo.VirAxisName.VirMain].Status.fActPos>=CamOutArgel  AND arrAxisCtrl[AxiseNo.VirAxisName.VirMain].Status.fActPos<=(CamOutArgel+5) THEN
		IF (Mach_Control.Ca_b.Ca_CacheBeltDLOK AND NOT fbCaCamInCarryingUpDown2OutCamFlge) OR Mach_Control.U.EmptyRunMode  THEN
			Mach_Control.Ca_b.Ca_CacheBelting:=TRUE;//f负极搬运升降取极片中	
			arrCyCtrl[arrCyNo.ElectValveName.CaCarryingVacuum2].Cmd.bON:=FALSE;//负极送片搬运真空开
			arrCyCtrl[arrCyNo.ElectValveName.CaCarryingVacuum2].Cmd.bOFF:=TRUE;//负极送片搬运真空开
		ELSE
			//arrCyCtrl[arrCyNo.ElectValveName.CaCarryingVacuum2].Cmd.bON:=FALSE;//负极送片搬运真空开
			fbCaCamInCarryingUpDown2.bCamInExecute:=FALSE;//负极升解除耦合
			Mach_Control.Ca_b.Ca_CacheBelting:=FALSE;
		END_IF								
	END_IF
	//解除负极搬运升降凸轮耦合标记
	fbCaCamInCarryingUpDown2OutCam_F_TRIG(CLK:=fbCaCamInCarryingUpDown2.bCamInExecute , Q=> );
	IF fbCaCamInCarryingUpDown2OutCam_F_TRIG.Q THEN
		fbCaCamInCarryingUpDown2OutCamFlge:=TRUE;//负极升降2凸轮解耦标记
	END_IF	
*)			
410:							
	//打开或关闭真空，标记对应位置有料
	IF 	arrAxisCtrl[AxiseNo.VirAxisName.VirMain].Status.fActPos>=234 THEN//198

		Mach_Control.An_b.An_Rectifydev_CS:=0;
		CCD.Over.Start.stPoleNo:=Par.stDT_date.An_MQ_Slice[2].stPoleNo;
	(*	
		arrCyCtrl[arrCyNo.ElectValveName.AnCarryingVacuum].Cmd.bOFF:=TRUE;//正极送片搬运真空关
		arrCyCtrl[arrCyNo.ElectValveName.AnCarryingVacuumBark].Cmd.bON:=TRUE;//正极送片搬运破真空开
		arrCyCtrl[arrCyNo.ElectValveName.AnDTCarryingVacuum].Cmd.bOFF:=TRUE;//正极叠片搬运真空关
		arrCyCtrl[arrCyNo.ElectValveName.AnDTCarryingVacuumBark].Cmd.bON:=TRUE;//正极叠片搬运破真空开
	*)	
		arrCyCtrl[arrCyNo.ElectValveName.AnCarryingVacuum].Cmd.bON:=FALSE;//正极送片搬运真空关
		arrCyCtrl[arrCyNo.ElectValveName.AnCarryingVacuum].Cmd.bOFF:=TRUE;//正极送片搬运真空关
		arrCyCtrl[arrCyNo.ElectValveName.AnCarryingVacuumBark].Cmd.bON:=TRUE;//正极送片搬运破真空开
		arrCyCtrl[arrCyNo.ElectValveName.AnCarryingVacuumBark].Cmd.bOFF:=FALSE;//正极送片搬运破真空开
		
		arrCyCtrl[arrCyNo.ElectValveName.AnDTCarryingVacuum].Cmd.bON:=FALSE;//正极送片搬运真空关
		arrCyCtrl[arrCyNo.ElectValveName.AnDTCarryingVacuum].Cmd.bOFF:=TRUE;//正极送片搬运真空关
		arrCyCtrl[arrCyNo.ElectValveName.AnDTCarryingVacuumBark].Cmd.bON:=TRUE;//正极送片搬运破真空开
		arrCyCtrl[arrCyNo.ElectValveName.AnDTCarryingVacuumBark].Cmd.bOFF:=FALSE;//正极送片搬运破真空开	
		
		arrCyCtrl[arrCyNo.ElectValveName.AndeviationVacuum].Cmd.bON:=TRUE;//正极纠偏平台真空开	
		arrCyCtrl[arrCyNo.ElectValveName.AndeviationVacuum].Cmd.bOFF:=FALSE;//正极纠偏平台真空开	

		Mach_Control.An_b.An_DPCarryingFalg :=FALSE;//复位正极叠片搬运吸盘上有料标记
		//IF Mach_Control.An_b.An_CarryingFalg THEN
			Mach_Control.An_b.An_deviationFalg:=TRUE;//置位纠偏平台上有料标记
			Mach_Control.An_b.An_CarryingFalg:=FALSE;//复位正极送片搬运吸盘上有料标记
		//END_IF
		
		Par.stDT_date.An_MQ_Slice[1]:=Par.stDT_date.An_MQ_Slice[0];
		
		(*
		IF (Mach_Control.Ca_b.Ca_CacheBelting AND NOT fbCaCamInCarryingUpDown2OutCamFlge) OR Mach_Control.U.EmptyRunMode  THEN
			Mach_Control.Ca_b.Ca_CarryingFalg:=TRUE;//复位负极送片搬运吸盘上有料标记
			Par.stDT_date.Ca_MQ_Slice[7]:=Par.stDT_date.Ca_MQ_Slice[6];
		END_IF*)
		
		
		arrAxisCtrl[AxiseNo.AxisName.CaCarryingUpDown2].Cmd.bStop:=FALSE;
	

		//判断负极纠偏台是否允许取料
		IF Ca_deviationDPOKFalg AND NOT DP_CheseCam AND iCaCamInSel2=1 THEN		
			arrCyCtrl[arrCyNo.ElectValveName.CaDTCarryingVacuum].Cmd.bON:=FALSE;//负极叠台搬运真空开	
			arrCyCtrl[arrCyNo.ElectValveName.CaDTCarryingVacuum].Cmd.bOFF:=TRUE;//负极叠台搬运真空开	
			arrCyCtrl[arrCyNo.ElectValveName.CadeviationVacuum].Cmd.bOFF:=TRUE;//负极纠偏平台真空关
			arrCyCtrl[arrCyNo.ElectValveName.CadeviationVacuum].Cmd.bON:=FALSE;//负极纠偏平台真空关
			arrCyCtrl[arrCyNo.ElectValveName.CadeviationVacuumBark].Cmd.bON:=TRUE;//负极纠偏平台破真空开	
			arrCyCtrl[arrCyNo.ElectValveName.CadeviationVacuumBark].Cmd.bOFF:=FALSE;//负极纠偏平台破真空开		
			//IF 	Mach_Control.Ca_b.Ca_deviationFalg THEN				
				Mach_Control.Ca_b.Ca_DPCarryingFalg :=TRUE;//置位负极叠片搬运吸盘上有料标记			
				Mach_Control.Ca_b.Ca_deviationFalg:=FALSE;//复位负极纠偏平台上有料标记	
			//END_IF			
			Par.stDT_date.Ca_MQ_Slice[9]:=Par.stDT_date.Ca_MQ_Slice[8];
		(*	
		ELSE   
			Ca_Step3:=10;//负极叠片搬运取纠偏台极片	
		*)	   
		END_IF									

		//判断正极纠偏台是否允许放料
		IF An_deviationFPOKFalg THEN			
			arrCyCtrl[arrCyNo.ElectValveName.AnCarryingVacuumBark].Cmd.bON:=TRUE;//正极送片搬运真空关
			arrCyCtrl[arrCyNo.ElectValveName.AnCarryingVacuumBark].Cmd.bOFF:=FALSE;//正极送片搬运破真空开
			arrCyCtrl[arrCyNo.ElectValveName.AndeviationVacuum].Cmd.bON:=TRUE;//正极纠偏平台真空开		
			arrCyCtrl[arrCyNo.ElectValveName.AndeviationVacuum].Cmd.bOFF:=FALSE;//正极纠偏平台真空开	
			//IF Mach_Control.An_b.An_CarryingFalg THEN	
				Mach_Control.An_b.An_deviationFalg:=TRUE;//置位正极纠偏平台上有料标记
				Mach_Control.An_b.An_CarryingFalg:=FALSE;//复位正极送片搬运吸盘上有料标记						
			//END_IF			
			Par.stDT_date.An_MQ_Slice[1]:=Par.stDT_date.An_MQ_Slice[0];//送片机械手传送至纠偏平台
		ELSE   
			An_Step1:=10;//正极送片搬运放片到纠偏台			   
		END_IF
	END_IF

		IF 	arrAxisCtrl[AxiseNo.VirAxisName.VirMain].Status.fActPos>=342 THEN//198
			CCD.Over.Start.iPliesNo:=UINT_TO_INT(Mach_Control.Ca_b.Ca_Quantited + Mach_Control.An_b.An_Quantited+1);	
			IF NOT An_Number THEN
				CCD.Over.Start.iPhotoDo:=1;
			ELSE
				CCD.Over.Start.iPhotoDo:=2;
			END_IF
			CCD.Over.Finish.OverhandResult:=0;
			Mach_Control.DT_b.CDD_OverStart:=TRUE;	
			IF NOT An_Number THEN
				DP_Step3:=6666;					
			END_IF
			
        END_IF
END_CASE



//判断主轴是否完成
CASE  DP_Step4 OF
100://叠负极主轴定位完成判断				
	IF arrAxis[AxiseNo.VirAxisName.VirMain].NcToPlc.SetPos=360 AND  arrAxis[AxiseNo.VirAxisName.VirMain].Status.NotMoving  THEN
		//如果，叠片搬运掉片报警就不计数		
		IF NOT Ca_Number THEN
			Mach_Control.Ca_b.Ca_Quantited:=Mach_Control.Ca_b.Ca_Quantited+1;
			DPcount:=DPcount+1;
			IF Mach_Control.U.EmptyRunMode THEN
				Mach_Control.Ca_b.Ca_EmptyRunKDQuantited:=Mach_Control.Ca_b.Ca_EmptyRunKDQuantited +1;
//			ELSE
//				Mach_Control.Ca_b.Ca_EmptyRunKDQuantited:=0;
			END_IF
			Par.stDT_date.YD_JS_L:=Par.stDT_date.YD_JS_L+1;
			Mach_Control.Ca_b.Ca_CCD_amount:=0;
				//叠台升降轴下降
				IF NOT Mach_Control.U.EmptyRunMode  THEN
					arrAxisCtrl[AxiseNo.AxisName.DTUpDown].Cmd.fPosition_of_Rel:=-(Par.stDT_date.Ca_Thickness+Par.stDT_date.SEPTA_Thickness+Par.stDT_date.Pole_ThicknessCom);
				ELSE
					arrAxisCtrl[AxiseNo.AxisName.DTUpDown].Cmd.fPosition_of_Rel:=-Par.stDT_date.SEPTA_Thickness;
				END_IF
				IF Mach_Control.Ca_b.Ca_Quantited + Mach_Control.An_b.An_Quantited>3 THEN
					arrAxisPar[AxiseNo.AxisName.DTUpDown].fVelocity_of_Rel:=100;
					arrAxisCtrl[AxiseNo.AxisName.DTUpDown].Cmd.bMoveRel:=TRUE;
				END_IF
		END_IF
		Mach_Control.An_b.An_CCDStart :=FALSE;//启动CCD拍照						
		DP_Step1:=100;//解除耦合，主轴回零子程序
		
		IF Mach_Control.DT_b.SinStepMode THEN//单步调试模式
			DP_SinStepe:=TRUE;
		ELSE
			DP_SinStepe:=FALSE;	
		END_IF
		
		DP_Step0:=0;
		Ca_AlarmTON[11].IN:=FALSE;
		IF Ca_Number  THEN
			DP_Step6:=6666;
		ELSIF Mach_Control.DT_b.DT_Overhang THEN
			DP_Step6:=102;
		ELSE
			DP_Step6:=101;
		END_IF	
		DP_Step4:=110;	
	END_IF;	
110:
	IF ((*Ca_deviationFPOKFalg OR*) Ca_Step1=6666 OR Ca_Step1=0) AND ((*An_deviationDPOKFalg OR *)An_Step3=6666 OR An_Step3=0)  
		AND ((An_Step0=6666 OR An_Step0=0) OR Mach_Control.An_b.An_Quantited=Par.stDT_date.An_Quantity )  THEN         
		DP_Step4:=6666;
		DP_Step0:=0;
		Ca_deviationFPOKFalg:=FALSE;
		An_deviationDPOKFalg:=FALSE;  
	END_IF



		
200:	//叠正极主轴定位完成判断
	IF arrAxis[AxiseNo.VirAxisName.VirMain].NcToPlc.SetPos>=200 AND  NOT fbCaCamInCarryingUpDown2.bCamInExecute  THEN
		(*
		IF NOT  arrAxisCtrl[AxiseNo.AxisName.CaCarryingUpDown2].Cmd.arrbRealPoint[4] THEN
			arrAxisCtrl[AxiseNo.AxisName.CaCarryingUpDown2].Cmd.iGoSetPos:=4;//移动至流水线上方
		ELSE
			arrAxisCtrl[AxiseNo.AxisName.CaCarryingUpDown2].Cmd.iGoSetPos:=0;//移动至流水线上方
		END_IF
		*)
		;
	END_IF
	
	IF arrAxis[AxiseNo.VirAxisName.VirMain].NcToPlc.SetPos=360 AND  arrAxis[AxiseNo.VirAxisName.VirMain].Status.NotMoving  THEN
		//如果，叠片搬运掉片报警就不计数				
		IF NOT An_Number THEN
			Mach_Control.An_b.An_Quantited:=Mach_Control.An_b.An_Quantited+1;
			DPcount:=DPcount+1;			
			IF Mach_Control.U.EmptyRunMode THEN
				Mach_Control.An_b.An_EmptyRunKDQuantited:=Mach_Control.An_b.An_EmptyRunKDQuantited +1;
//			ELSE
//				Mach_Control.An_b.An_EmptyRunKDQuantited:=0;
			END_IF
			Par.stDT_date.YD_JS_R:=Par.stDT_date.YD_JS_R+1;
			Mach_Control.An_b.An_CCD_amount:=0;
			//叠台升降轴下降
			IF NOT Mach_Control.U.EmptyRunMode  THEN
					arrAxisCtrl[AxiseNo.AxisName.DTUpDown].Cmd.fPosition_of_Rel:=-(Par.stDT_date.An_Thickness+Par.stDT_date.SEPTA_Thickness+Par.stDT_date.Pole_ThicknessCom);
			ELSE
					arrAxisCtrl[AxiseNo.AxisName.DTUpDown].Cmd.fPosition_of_Rel:=-Par.stDT_date.SEPTA_Thickness;
			END_IF
			IF Mach_Control.Ca_b.Ca_Quantited + Mach_Control.An_b.An_Quantited>3 THEN
					arrAxisPar[AxiseNo.AxisName.DTUpDown].fVelocity_of_Rel:=100;
					arrAxisCtrl[AxiseNo.AxisName.DTUpDown].Cmd.bMoveRel:=TRUE;
			END_IF	
		END_IF
		Mach_Control.Ca_b.Ca_CCDStart :=FALSE;//启动CCD拍照			
		DP_Step1:=100;//解除耦合，主轴回零	

		(*
		IF  (Mach_Control.Ca_b.Ca_CacheBelting AND NOT fbCaCamInCarryingUpDown2OutCamFlge) OR Mach_Control.U.EmptyRunMode  THEN
			Par.stDT_date.Ca_betlCount.5:=FALSE;//复位负极流水线极片标记
			Mach_Control.Ca_b.Ca_CacheBelting:=FALSE;
		END_IF	*)
	
						
		arrCyCtrl[arrCyNo.ElectValveName.CadeviationVacuumBark].Cmd.bOFF:=TRUE;//负极纠偏平台破真空关	
		IF Mach_Control.DT_b.SinStepMode THEN//单步调试模式
			DP_SinStepe:=TRUE;
		ELSE
			DP_SinStepe:=FALSE;	
		END_IF							
		DP_Step0:=0;
		An_AlarmTON[11].IN:=FALSE;
		IF An_Number THEN
			  DP_Step7:=6666;
		ELSIF  Mach_Control.DT_b.DT_Overhang THEN
			  DP_Step7:=202;
		ELSE
			  DP_Step7:=201;
		END_IF
		DP_Step4:=210;	
		(*	
			IF  Mach_Control.DT_b.DT_Overhang AND NOT An_Number THEN
				  DP_Step7:=202;
			ELSIF An_Number THEN
				  DP_Step7:=6666;
			ELSE
				  DP_Step7:=201;
			END_IF
			DP_Step4:=6666;	
		*)
	END_IF;	
210:
	IF ((*An_deviationFPOKFalg OR *)An_Step1=6666 OR An_Step1=0) AND ((*Ca_deviationDPOKFalg OR *)Ca_Step3=6666 OR Ca_Step3=0) 
	AND (Ca_Step0=6666 OR Ca_Step0=0) THEN          
		DP_Step4:=6666;
		DP_Step0:=0;
		An_deviationFPOKFalg:=FALSE;
		Ca_deviationDPOKFalg:=FALSE; 
	END_IF

			
END_CASE



//观察NG片用，发现问题后删除
IF Ca_NGTest1.Q THEN
	Ca_NG:=Ca_NG+1;
END_IF


CASE  DP_Step5 OF
100://判断主轴运行时负极叠片搬运升降真空报警
	IF arrAxisCtrl[AxiseNo.VirAxisName.VirMain].Status.fActPos>0 AND arrAxisCtrl[AxiseNo.VirAxisName.VirMain].Status.fActPos<220 THEN
		IF Ca_Number THEN	
			DP_Step5:=110;
			arrCyCtrl[arrCyNo.ElectValveName.CaDTCarryingVacuum].Cmd.bON:=TRUE;//负极叠片搬运破真空开	
			arrCyCtrl[arrCyNo.ElectValveName.CaDTCarryingVacuum].Cmd.bOFF:=FALSE;//负极叠片搬运破真空开	
		END_IF
		Ca_NGTest1(CLK:=(CCD.CaRec.Finish.RectifyResult=2) , Q=> );
	ELSE 
		DP_Step5:=6666;
	END_IF

110:
	fbCaCamInDTCarryingUpDown.bCamInExecute:=FALSE;//负极叠片搬运升降
	fbCamInLeftYDUpDown.bCamInExecute:=FALSE;//左压刀升降
	fbCamInLeftYDLine.bCamInExecute:=FALSE;//左压刀开合
	IF NOT  fbCaCamInDTCarryingUpDown.bCamInExecute AND NOT fbCamInLeftYDUpDown.bCamInExecute AND NOT  fbCamInLeftYDLine.bCamInExecute THEN
		DP_Step5:=120;
		arrCyCtrl[arrCyNo.ElectValveName.CaDTCarryingVacuum].Cmd.bON:=FALSE;//负极叠片搬运真空开
		arrCyCtrl[arrCyNo.ElectValveName.CaDTCarryingVacuum].Cmd.bOFF:=TRUE;//负极叠片搬运真空开
	END_IF

120:
	arrAxisCtrl[AxiseNo.AxisName.CaDTCarryingUpDown].Cmd.bGearOut:=TRUE;
	arrAxisCtrl[AxiseNo.AxisName.LeftYDLine].Cmd.bGearOut:=TRUE;
	arrAxisCtrl[AxiseNo.AxisName.LeftYDUpDown].Cmd.bGearOut:=TRUE;
	IF NOT arrAxisCtrl[AxiseNo.AxisName.CaDTCarryingUpDown].Status.Coupled AND NOT arrAxisCtrl[AxiseNo.AxisName.LeftYDLine].Status.Coupled
	AND NOT arrAxisCtrl[AxiseNo.AxisName.LeftYDUpDown].Status.Coupled THEN
		arrAxisCtrl[AxiseNo.AxisName.CaDTCarryingUpDown].Cmd.bGearOut:=FALSE;
		arrAxisCtrl[AxiseNo.AxisName.LeftYDLine].Cmd.bGearOut:=FALSE;
		arrAxisCtrl[AxiseNo.AxisName.LeftYDUpDown].Cmd.bGearOut:=FALSE;
		DP_Step5:=130;
	END_IF

130:
	IF arrAxisCtrl[AxiseNo.AxisName.CaDTCarryingUpDown].Status.Homed AND arrAxisCtrl[AxiseNo.AxisName.CaDTCarryingUpDown].Status.NoMoving AND 
		NOT arrAxisCtrl[AxiseNo.AxisName.CaDTCarryingUpDown].Status.Error THEN
		IF arrAxisCtrl[AxiseNo.AxisName.CaDTCarryingUpDown].Cmd.arrbRealPoint[4] THEN
			arrCyCtrl[arrCyNo.ElectValveName.CaDTCarryingVacuum].Cmd.bON:=FALSE;//负极叠片搬运真空开
			arrCyCtrl[arrCyNo.ElectValveName.CaDTCarryingVacuum].Cmd.bOFF:=TRUE;//负极叠片搬运真空开
			arrAxisCtrl[AxiseNo.AxisName.CaDTCarryingUpDown].Cmd.iGoSetPos:=0;
			DP_Step5:=6666;
		ELSE
			arrAxisCtrl[AxiseNo.AxisName.CaDTCarryingUpDown].Cmd.iGoSetPos:=4;//负极叠片升降移动至等待高度
		END_IF
	END_IF







200://判断主轴运行时正极叠片搬运升降真空报警
	IF arrAxisCtrl[AxiseNo.VirAxisName.VirMain].Status.fActPos>0 AND arrAxisCtrl[AxiseNo.VirAxisName.VirMain].Status.fActPos<220 THEN
		IF An_Number THEN	
			DP_Step5:=210;
			arrCyCtrl[arrCyNo.ElectValveName.AnDTCarryingVacuumBark].Cmd.bON:=TRUE;//正极叠片搬运破真空开	
		END_IF
	ELSE 
		DP_Step5:=6666;
	END_IF

210:
	fbAnCamInDTCarryingUpDown.bCamInExecute:=FALSE;//正极叠片搬运升降
	fbCamInRightYDUpDown.bCamInExecute:=FALSE;
	fbCamInRightYDLine.bCamInExecute:=FALSE;
	IF NOT fbAnCamInDTCarryingUpDown.bCamInExecute AND NOT fbCamInRightYDUpDown.bCamInExecute AND NOT fbCamInRightYDLine.bCamInExecute THEN
		DP_Step5:=220;
		arrCyCtrl[arrCyNo.ElectValveName.AnDTCarryingVacuumBark].Cmd.bON:=FALSE;//正极叠片搬运破真空关	
	END_IF
220:
	arrAxisCtrl[AxiseNo.AxisName.AnDTCarryingUpDown].Cmd.bGearOut:=TRUE;
	arrAxisCtrl[AxiseNo.AxisName.RightYDLine].Cmd.bGearOut:=TRUE;
	arrAxisCtrl[AxiseNo.AxisName.RightYDUpDown].Cmd.bGearOut:=TRUE;
	IF NOT arrAxisCtrl[AxiseNo.AxisName.AnDTCarryingUpDown].Status.Coupled AND NOT arrAxisCtrl[AxiseNo.AxisName.RightYDLine].Status.Coupled AND
		NOT arrAxisCtrl[AxiseNo.AxisName.RightYDUpDown].Status.Coupled  THEN
		arrAxisCtrl[AxiseNo.AxisName.AnDTCarryingUpDown].Cmd.bGearOut:=FALSE;
		arrAxisCtrl[AxiseNo.AxisName.RightYDLine].Cmd.bGearOut:=FALSE;
		arrAxisCtrl[AxiseNo.AxisName.RightYDUpDown].Cmd.bGearOut:=FALSE;
		DP_Step5:=230;
	END_IF

230:
	IF arrAxisCtrl[AxiseNo.AxisName.AnDTCarryingUpDown].Status.Homed AND arrAxisCtrl[AxiseNo.AxisName.AnDTCarryingUpDown].Status.NoMoving AND 
	NOT arrAxisCtrl[AxiseNo.AxisName.AnDTCarryingUpDown].Status.Error THEN
		IF arrAxisCtrl[AxiseNo.AxisName.AnDTCarryingUpDown].Cmd.arrbRealPoint[4] THEN
			arrAxisCtrl[AxiseNo.AxisName.AnDTCarryingUpDown].Cmd.iGoSetPos:=0;
			DP_Step5:=6666;
		ELSE
			arrAxisCtrl[AxiseNo.AxisName.AnDTCarryingUpDown].Cmd.iGoSetPos:=4;//正极叠片升降移动至等待高度
		END_IF
	END_IF
		
END_CASE




CASE DP_Step6 OF
101:
	IF (CCD.Over.Finish.OverhandResult=4 OR CCD.Over.Finish.OverhandResult=2 OR CCD.Over.Finish.OverhandResult=1 ) AND NOT Ca_Number 
		AND( (arrAxisCtrl[AxiseNo.VirAxisName.VirMain].Status.fActPos>100 AND  arrAxisCtrl[AxiseNo.VirAxisName.VirMain].Status.fActPos<220) OR (arrAxisCtrl[AxiseNo.VirAxisName.VirMain].Status.fActPos=360)) THEN		
		DP_Step6:=102;
	ELSIF Ca_Number OR Mach_Control.U.EmptyRunMode OR Mach_Control.DT_b.DT_Overhang THEN//负极报警，空跑模式，Overhang屏蔽直接跳过
		DP_Step6:=6666;
	ELSIF NOT Ca_Number AND arrAxisCtrl[AxiseNo.VirAxisName.VirMain].Status.fActPos>220 AND arrAxisCtrl[AxiseNo.VirAxisName.VirMain].Status.fActPos<360 
		AND  CCD.Over.Finish.OverhandResult=0   THEN
		Mach_Control.Ca_b.Error[25]:=TRUE;//负极极片对齐度检测返回结果超时
		Par.stDT_date.Overhang_CSJS:=Par.stDT_date.Overhang_CSJS+1;
		DP_Step6:=6666;
	ELSIF CCD.Over.Finish.OverhandResult=3   THEN		
		Mach_Control.Ca_b.Error[27]:=TRUE;  //负极极片对齐度检测返回结果无片报警
		DP_Step6:=102;
	END_IF
					
102:
	CellMemory[Mach_Control.DT_b.DT_Memory].Overhang_Result[CCD.Over.Start.iPliesNo]:=CCD.Over.Finish.OverhandResult;
	CellMemory[Mach_Control.DT_b.DT_Memory].DiaphragmUnwindingTension2[CCD.Over.Start.iPliesNo]:=LIMIT(150,ABS(Mach_Control.DT_b.DiaphragmUnwindingTension),250);	
	CellMemory[Mach_Control.DT_b.DT_Memory].Ca_Ear_Overhang_A_C[Mach_Control.Ca_b.Ca_Quantited]:=ABS(CCD.Over.Finish.AnCaOverhandX1);
	CellMemory[Mach_Control.DT_b.DT_Memory].Ca_Ear_Overhang_S_CIL[Mach_Control.Ca_b.Ca_Quantited]:=ABS(CCD.Over.Finish.PoleOverhandX1);
	CellMemory[Mach_Control.DT_b.DT_Memory].Ca_Ear_No_Overhang_A_C[Mach_Control.Ca_b.Ca_Quantited]:=ABS(CCD.Over.Finish.AnCaOverhandX4);
	CellMemory[Mach_Control.DT_b.DT_Memory].Ca_Ear_No_Overhang_S_A[Mach_Control.Ca_b.Ca_Quantited]:=ABS(CCD.Over.Finish.PoleOverhandX4);
	
	CellMemory[Mach_Control.DT_b.DT_Memory].Ca_Ear_L_Overhang_A_C[Mach_Control.Ca_b.Ca_Quantited]:=ABS(CCD.Over.Finish.AnCaOverhandY1);
	CellMemory[Mach_Control.DT_b.DT_Memory].Ca_Ear_L_Overhang_S_A[Mach_Control.Ca_b.Ca_Quantited]:=ABS(CCD.Over.Finish.PoleOverhandY1);
	CellMemory[Mach_Control.DT_b.DT_Memory].Ca_Ear_R_Overhang_A_C[Mach_Control.Ca_b.Ca_Quantited]:=ABS(CCD.Over.Finish.AnCaOverhandY4);
	CellMemory[Mach_Control.DT_b.DT_Memory].Ca_Ear_R_Overhang_S_A[Mach_Control.Ca_b.Ca_Quantited]:=ABS(CCD.Over.Finish.PoleOverhandY4);
	
	CellMemory[Mach_Control.DT_b.DT_Memory].Ca_Cell_Overhang:=ABS(CCD.Over.Finish.AddOverhangX1);
	CellMemory[Mach_Control.DT_b.DT_Memory].Ca_Cell_Overhang_No:=ABS(CCD.Over.Finish.AddOverhangX4);
	CellMemory[Mach_Control.DT_b.DT_Memory].Ca_Cell_Overhang_L:=ABS(CCD.Over.Finish.AddOverhangY1);
	CellMemory[Mach_Control.DT_b.DT_Memory].Ca_Cell_Overhang_R:=ABS(CCD.Over.Finish.AddOverhangY4);
	
	CellMemory[Mach_Control.DT_b.DT_Memory].Ca_PoleOverhandX2[Mach_Control.Ca_b.Ca_Quantited]:=ABS(CCD.Over.Finish.PoleOverhandX2);
	CellMemory[Mach_Control.DT_b.DT_Memory].Ca_PoleOverhandX3[Mach_Control.Ca_b.Ca_Quantited]:=ABS(CCD.Over.Finish.PoleOverhandX3);
	CellMemory[Mach_Control.DT_b.DT_Memory].Ca_PoleOverhandY2[Mach_Control.Ca_b.Ca_Quantited]:=ABS(CCD.Over.Finish.PoleOverhandY2);
	CellMemory[Mach_Control.DT_b.DT_Memory].Ca_PoleOverhandY3[Mach_Control.Ca_b.Ca_Quantited]:=ABS(CCD.Over.Finish.PoleOverhandY3);
	
	CellMemory[Mach_Control.DT_b.DT_Memory].Ca_AnCaOverhandX2[Mach_Control.Ca_b.Ca_Quantited]:=ABS(CCD.Over.Finish.AnCaOverhandX2);
	CellMemory[Mach_Control.DT_b.DT_Memory].Ca_AnCaOverhandX3[Mach_Control.Ca_b.Ca_Quantited]:=ABS(CCD.Over.Finish.AnCaOverhandX3);
	CellMemory[Mach_Control.DT_b.DT_Memory].Ca_AnCaOverhandY2[Mach_Control.Ca_b.Ca_Quantited]:=ABS(CCD.Over.Finish.AnCaOverhandY2);
	CellMemory[Mach_Control.DT_b.DT_Memory].Ca_AnCaOverhandY3[Mach_Control.Ca_b.Ca_Quantited]:=ABS(CCD.Over.Finish.AnCaOverhandY3);
	
	CellMemory[Mach_Control.DT_b.DT_Memory].Ca_AddOverhangX2:=ABS(CCD.Over.Finish.AddOverhangX2);
	CellMemory[Mach_Control.DT_b.DT_Memory].Ca_AddOverhangX3:=ABS(CCD.Over.Finish.AddOverhangX3);
	CellMemory[Mach_Control.DT_b.DT_Memory].Ca_AddOverhangY2:=ABS(CCD.Over.Finish.AddOverhangY2);
	CellMemory[Mach_Control.DT_b.DT_Memory].Ca_AddOverhangY3:=ABS(CCD.Over.Finish.AddOverhangY3);
	
	CellMemory[Mach_Control.DT_b.DT_Memory].Ca_MQ_Slice[Mach_Control.Ca_b.Ca_Quantited]:=Par.stDT_date.Ca_MQ_Slice[9];
	Ca_AlarmTON[11].IN:=FALSE;
	DP_Step6:=103;	


103:
	CCD.Over.Finish.OverhandResult:=0;
	DP_Step6:=6666;	


END_CASE







CASE DP_Step7 OF
201:
	IF (CCD.Over.Finish.OverhandResult=4 OR CCD.Over.Finish.OverhandResult=2 OR CCD.Over.Finish.OverhandResult=1 ) AND NOT An_Number 
		AND ((arrAxisCtrl[AxiseNo.VirAxisName.VirMain].Status.fActPos>100 AND  arrAxisCtrl[AxiseNo.VirAxisName.VirMain].Status.fActPos<220) OR
		 (arrAxisCtrl[AxiseNo.VirAxisName.VirMain].Status.fActPos=360))THEN
		DP_Step7:=202;
	ELSIF An_Number OR Mach_Control.U.EmptyRunMode OR Mach_Control.DT_b.DT_Overhang THEN//负极报警，空跑模式，Overhang屏蔽直接跳过
		DP_Step7:=6666;	
	ELSIF   NOT An_Number AND arrAxisCtrl[AxiseNo.VirAxisName.VirMain].Status.fActPos>220 AND arrAxisCtrl[AxiseNo.VirAxisName.VirMain].Status.fActPos<360 
		AND CCD.Over.Finish.OverhandResult=0 THEN
		Mach_Control.An_b.Error[25]:=TRUE;//正极极片对齐度检测返回结果超时
		Par.stDT_date.Overhang_CSJS:=Par.stDT_date.Overhang_CSJS+1;
		DP_Step7:=6666;	
	ELSIF CCD.Over.Finish.OverhandResult=3 THEN 		
		Mach_Control.An_b.Error[27]:=TRUE; //正极极片对齐度检测返回结果无片报警
		DP_Step7:=202;	
	END_IF
							
											
202:
	CellMemory[Mach_Control.DT_b.DT_Memory].Overhang_Result[CCD.Over.Start.iPliesNo]:=CCD.Over.Finish.OverhandResult;	
	CellMemory[Mach_Control.DT_b.DT_Memory].DiaphragmUnwindingTension2[CCD.Over.Start.iPliesNo]:=LIMIT(150,ABS(Mach_Control.DT_b.DiaphragmUnwindingTension),250);
	CellMemory[Mach_Control.DT_b.DT_Memory].An_Ear_Overhang_A_C[Mach_Control.An_b.An_Quantited]:=ABS(CCD.Over.Finish.AnCaOverhandX1);
	CellMemory[Mach_Control.DT_b.DT_Memory].An_Ear_Overhang_S_CIL[Mach_Control.An_b.An_Quantited]:=ABS(CCD.Over.Finish.PoleOverhandX1);
	CellMemory[Mach_Control.DT_b.DT_Memory].An_Ear_No_Overhang_A_C[Mach_Control.An_b.An_Quantited]:=ABS(CCD.Over.Finish.AnCaOverhandX4);
	CellMemory[Mach_Control.DT_b.DT_Memory].An_Ear_No_Overhang_S_A[Mach_Control.An_b.An_Quantited]:=ABS(CCD.Over.Finish.PoleOverhandX4);
	
	CellMemory[Mach_Control.DT_b.DT_Memory].An_Ear_L_Overhang_A_C[Mach_Control.An_b.An_Quantited]:=ABS(CCD.Over.Finish.AnCaOverhandY1);
	CellMemory[Mach_Control.DT_b.DT_Memory].An_Ear_L_Overhang_S_A[Mach_Control.An_b.An_Quantited]:=ABS(CCD.Over.Finish.PoleOverhandY1);
	CellMemory[Mach_Control.DT_b.DT_Memory].An_Ear_R_Overhang_A_C[Mach_Control.An_b.An_Quantited]:=ABS(CCD.Over.Finish.AnCaOverhandY4);
	CellMemory[Mach_Control.DT_b.DT_Memory].An_Ear_R_Overhang_S_A[Mach_Control.An_b.An_Quantited]:=ABS(CCD.Over.Finish.PoleOverhandY4);
	
	CellMemory[Mach_Control.DT_b.DT_Memory].An_Cell_Overhang:=ABS(CCD.Over.Finish.AddOverhangX1);
	CellMemory[Mach_Control.DT_b.DT_Memory].An_Cell_Overhang_No:=ABS(CCD.Over.Finish.AddOverhangX4);
	CellMemory[Mach_Control.DT_b.DT_Memory].An_Cell_Overhang_L:=ABS(CCD.Over.Finish.AddOverhangY1);
	CellMemory[Mach_Control.DT_b.DT_Memory].An_Cell_Overhang_R:=ABS(CCD.Over.Finish.AddOverhangY4);
	
	CellMemory[Mach_Control.DT_b.DT_Memory].An_PoleOverhandX2[Mach_Control.An_b.An_Quantited]:=ABS(CCD.Over.Finish.PoleOverhandX2);
	CellMemory[Mach_Control.DT_b.DT_Memory].An_PoleOverhandX3[Mach_Control.An_b.An_Quantited]:=ABS(CCD.Over.Finish.PoleOverhandX3);
	CellMemory[Mach_Control.DT_b.DT_Memory].An_PoleOverhandY2[Mach_Control.An_b.An_Quantited]:=ABS(CCD.Over.Finish.PoleOverhandY2);
	CellMemory[Mach_Control.DT_b.DT_Memory].An_PoleOverhandY3[Mach_Control.An_b.An_Quantited]:=ABS(CCD.Over.Finish.PoleOverhandY3);
	
	CellMemory[Mach_Control.DT_b.DT_Memory].An_AnCaOverhandX2[Mach_Control.An_b.An_Quantited]:=ABS(CCD.Over.Finish.AnCaOverhandX2);
	CellMemory[Mach_Control.DT_b.DT_Memory].An_AnCaOverhandX3[Mach_Control.An_b.An_Quantited]:=ABS(CCD.Over.Finish.AnCaOverhandX3);
	CellMemory[Mach_Control.DT_b.DT_Memory].An_AnCaOverhandY2[Mach_Control.An_b.An_Quantited]:=ABS(CCD.Over.Finish.AnCaOverhandY2);
	CellMemory[Mach_Control.DT_b.DT_Memory].An_AnCaOverhandY3[Mach_Control.An_b.An_Quantited]:=ABS(CCD.Over.Finish.AnCaOverhandY3);
	
	CellMemory[Mach_Control.DT_b.DT_Memory].An_AddOverhangX2:=ABS(CCD.Over.Finish.AddOverhangX2);
	CellMemory[Mach_Control.DT_b.DT_Memory].An_AddOverhangX3:=ABS(CCD.Over.Finish.AddOverhangX3);
	CellMemory[Mach_Control.DT_b.DT_Memory].An_AddOverhangY2:=ABS(CCD.Over.Finish.AddOverhangY2);
	CellMemory[Mach_Control.DT_b.DT_Memory].An_AddOverhangY3:=ABS(CCD.Over.Finish.AddOverhangY3);
	
	CellMemory[Mach_Control.DT_b.DT_Memory].An_MQ_Slice[Mach_Control.An_b.An_Quantited]:=Par.stDT_date.An_MQ_Slice[2];
	DP_Step7:=203;	

203:
	CCD.Over.Finish.OverhandResult:=0;
	DP_Step7:=6666;

END_CASE



CASE DP_Step8 OF	
100:
	Ca_StandbySub3_ton[2].IN:=FALSE;
	IF  NOT Mach_Control.U.CCD_ChosesHMI  AND NOT  Mach_Control.U.EmptyRunMode  THEN
		//IF arrAxis[AxiseNo.VirAxisName.VirMain].NcToPlc.SetPos>109 AND arrAxis[AxiseNo.VirAxisName.VirMain].NcToPlc.SetPos<=112   THEN
		IF arrAxis[AxiseNo.VirAxisName.VirMain].NcToPlc.SetPos>110 AND arrAxis[AxiseNo.VirAxisName.VirMain].NcToPlc.SetPos<=115   THEN
				CCD.CaRec.Finish.RectifyX1:=0;
				CCD.CaRec.Finish.RectifyX2:=0;
				CCD.CaRec.Finish.RectifyY:=0;		
				CCD.CaRec.Finish.RectifyResult:=0;//拍照结果清零									
				Mach_Control.Ca_b.Ca_CCDStart :=TRUE;//启动CCD拍照
				CCD.CaRec.Start.iPhotoDo:=1;//启动CCD第二次拍照
				//arrCyCtrl[arrCyNo.ElectValveName.CadeviationIonizedWind].Cmd.bON:=TRUE;//负极纠偏平台除尘
				//arrCyCtrl[arrCyNo.ElectValveName.AndeviationIonizedWind].Cmd.bON:=TRUE;//正极纠偏平台除尘
				DP_Step8:=110;
		END_IF
	ELSE
		DP_Step8:=6661;
	END_IF
110:
	Ca_StandbySub3_ton[2].IN:=CCD.CaRec.Finish.RectifyResult=0;
	IF Ca_StandbySub3_ton[2].Q THEN
		Mach_Control.DT_b.Error[51]:=TRUE;//检测负极纠偏平台空片结果返回超时
		DP_Step8:=9991;
	ELSIF CCD.CaRec.Finish.RectifyResult<>0 AND CCD.CaRec.Finish.RectifyResult<>3   THEN
		Mach_Control.Ca_b.Error[24]:=TRUE;//负极纠偏平台NG片未排掉报警，请拿掉
		Ca_StandbySub3_ton[2].IN:=FALSE;
		DP_Step8:=9992;
	ELSIF CCD.CaRec.Finish.RectifyResult=3  THEN
		DP_Step8:=6661;
	END_IF

200:
	An_StandbySub3_ton[2].IN:=FALSE;
	IF  NOT Mach_Control.U.CCD_ChosesHMI  AND NOT  Mach_Control.U.EmptyRunMode    THEN
		//IF arrAxis[AxiseNo.VirAxisName.VirMain].NcToPlc.SetPos>118 AND arrAxis[AxiseNo.VirAxisName.VirMain].NcToPlc.SetPos<=123  THEN
		IF arrAxis[AxiseNo.VirAxisName.VirMain].NcToPlc.SetPos>110 AND arrAxis[AxiseNo.VirAxisName.VirMain].NcToPlc.SetPos<=115   THEN
			CCD.AnRec.Finish.RectifyResult:=0;
			CCD.AnRec.Finish.RectifyX1:=0;
			CCD.AnRec.Finish.RectifyX2:=0;
			CCD.AnRec.Finish.RectifyY:=0;												
			Mach_Control.An_b.An_CCDStart :=TRUE;//启动CCD拍照
			CCD.AnRec.Start.iPhotoDo:=1;//第二次拍照
			//arrCyCtrl[arrCyNo.ElectValveName.CadeviationIonizedWind].Cmd.bON:=TRUE;//负极纠偏平台除尘
			//arrCyCtrl[arrCyNo.ElectValveName.AndeviationIonizedWind].Cmd.bON:=TRUE;//正极纠偏平台除尘
			DP_Step8:=210;
		END_IF
	ELSE
		DP_Step8:=6662;
	END_IF	
210:
	An_StandbySub3_ton[2].IN:=CCD.AnRec.Finish.RectifyResult=0;
	IF An_StandbySub3_ton[2].Q THEN				
		Mach_Control.DT_b.Error[52]:=TRUE;//检测正极纠偏平台空片结果返回超时
		An_StandbySub3_ton[2].IN:=FALSE;
		DP_Step8:=9993;		
	ELSIF CCD.AnRec.Finish.RectifyResult<>0 AND CCD.AnRec.Finish.RectifyResult<>3 THEN
		Mach_Control.An_b.Error[24]:=TRUE;//正极纠偏平台NG片未排掉报警，请拿掉 
		An_StandbySub3_ton[2].IN:=FALSE;
		DP_Step8:=9994;
	ELSIF CCD.AnRec.Finish.RectifyResult=3 THEN
		An_StandbySub3_ton[2].IN:=FALSE;
		DP_Step8:=6662;
	END_IF
	
END_CASE

*)
END_ACTION

ACTION _01DT_Auto3:

(*******************************************************************************************************叠完片后，空叠片隔膜***************************************************************************************************************************)
DT_TON[5](IN:= , PT:=T#300MS , Q=> , ET=> );//

IF Mach_Control.U.DT_iMode=1 THEN//在自动状态下
CASE DP_Step0 OF    //空叠隔膜流程
1000://判断主轴是否停止、是否在初始位、是否有轴在耦合中
	IF NOT DP_SinStepe THEN
		IF arrAxisCtrl[AxiseNo.VirAxisName.VirMain].Status.NoMoving AND arrAxisCtrl[AxiseNo.VirAxisName.VirMain].Status.fSetPos=0 AND NOT DT_AxiseCoupling THEN
			KD_Mark:=TRUE;//空叠隔膜中
			IF Mach_Control.DT_b.SinStepMode THEN//单步调试模式
				DP_SinStepe:=TRUE;
			ELSE
				DP_SinStepe:=FALSE;	
			END_IF
			DP_Step0:=1020;
		ELSE
			DP_Step1:=100;//解除耦合，主轴回零
			DP_Step0:=1010;
		END_IF
	END_IF
1010://判断主轴当前的当前位置是否为0
	IF DP_Step1=6666 AND arrAxisCtrl[AxiseNo.VirAxisName.VirMain].Status.NoMoving AND arrAxisCtrl[AxiseNo.VirAxisName.VirMain].Status.fSetPos=0 AND NOT DT_AxiseCoupling THEN
		IF Mach_Control.DT_b.SinStepMode THEN//单步调试模式
			DP_SinStepe:=TRUE;
		ELSE
			DP_SinStepe:=FALSE;	
		END_IF									
		DP_Step0:=1020;
	END_IF	

1020://判断NG气缸是否在安全位
	IF arrCyCtrl[arrCyNo.CylinderName.AnScrapbinCy].Status.ONState AND arrCyCtrl[arrCyNo.CylinderName.CaScrapbinUDCy].Status.OFFState AND
		arrCyCtrl[arrCyNo.CylinderName.CaScrapbinCy].Status.ONState AND arrCyCtrl[arrCyNo.CylinderName.PreDiaph].Status.OFFState AND 
		arrCyCtrl[arrCyNo.CylinderName.PoleHotCutterCy].Status.OFFState AND arrCyCtrl[arrCyNo.CylinderName.PoleTapeCy].Status.OFFState AND
		arrCyCtrl[arrCyNo.CylinderName.PoleTapeSplicerRCy].Status.ONState AND arrCyCtrl[arrCyNo.CylinderName.PoleTapeSplicerLCy].Status.ONState THEN
		DP_Step0:=1050;		
	ELSE
		DP_Step0:=1030;	
	END_IF
1030:
	arrCyCtrl[arrCyNo.CylinderName.AnScrapbinCy].Cmd.bON:=TRUE;
	arrCyCtrl[arrCyNo.CylinderName.PreDiaph].Cmd.bOFF:=TRUE;
	arrCyCtrl[arrCyNo.CylinderName.PoleHotCutterCy].Cmd.bOFF:=TRUE;
	arrCyCtrl[arrCyNo.CylinderName.PoleTapeCy].Cmd.bOFF:=TRUE;
	arrCyCtrl[arrCyNo.CylinderName.PoleTapeSplicerRCy].Cmd.bON:=TRUE;
	arrCyCtrl[arrCyNo.CylinderName.PoleTapeSplicerLCy].Cmd.bON:=TRUE;
	arrCyCtrl[arrCyNo.CylinderName.CaScrapbinCy].Cmd.bON:=TRUE;
	IF   arrCyCtrl[arrCyNo.CylinderName.AnScrapbinCy].Status.ONState AND  arrCyCtrl[arrCyNo.CylinderName.PreDiaph].Status.OFFState AND 
	arrCyCtrl[arrCyNo.CylinderName.PoleHotCutterCy].Status.OFFState AND arrCyCtrl[arrCyNo.CylinderName.PoleTapeCy].Status.OFFState AND
	arrCyCtrl[arrCyNo.CylinderName.PoleTapeSplicerRCy].Status.ONState AND arrCyCtrl[arrCyNo.CylinderName.PoleTapeSplicerLCy].Status.ONState
	AND arrCyCtrl[arrCyNo.CylinderName.CaScrapbinCy].Cmd.bON THEN
		DP_Step0:=1040;									
	END_IF
1040:
	arrCyCtrl[arrCyNo.CylinderName.CaScrapbinUDCy].Cmd.bOFF:=TRUE;
	IF  arrCyCtrl[arrCyNo.CylinderName.CaScrapbinUDCy].Status.OFFState THEN
		DP_Step0:=1050;	
	END_IF						
1050://	最后一层为负极片，所以，最开始先叠正极的隔膜
	KD_Mark:=TRUE;//空叠隔膜中
	IF NOT Bnt_Blueflaging THEN
		IF Mach_Control.An_b.An_KDQuantited  = Mach_Control.Ca_b.Ca_KDQuantited   THEN//先叠正极
			DP_Step0:=1100;
		ELSIF Mach_Control.An_b.An_KDQuantited  > Mach_Control.Ca_b.Ca_KDQuantited   THEN//先叠负极
			DP_Step0:=1500;
		END_IF
	ELSE//判断隔膜平移轴位置
		IF AN_CarryingPos1 THEN	
			DP_Step0:=1100;			
		ELSIF Ca_CarryingPos1 THEN
			DP_Step0:=1500;	
		ELSE
			Mach_Control.DT_b.Error[57]:=TRUE;//空叠隔膜时正负极都不在取片位	
		END_IF	
	(*
		IF (Mach_Control.An_b.An_KDQuantited  <= Mach_Control.Ca_b.Ca_KDQuantited) AND AN_CarryingPos1   THEN//先叠正极
			DP_Step0:=1100;
		ELSE 
			IF Ca_CarryingPos1 THEN	
				DP_Step0:=1500;	
			ELSE
				;//空叠隔膜时正负极都不在取片位	
			END_IF
		END_IF
	*)
	END_IF		

1100://判断叠台搬运机械手是否有片
	IF AN_CarryingPos1  THEN//正极搬运、叠片各轴在初始位	
		IF arrCyCtrl[arrCyNo.ElectValveName.AnDTCarryingVacuum].Io.DIOnSwitch AND  Mach_Control.An_b.An_DPCarryingFalg THEN//正极再取片位且叠台搬运有片,把当前片放到纠偏台
			DP_Step0:=1150;
		ELSE
			DP_Step0:=2000;	
		END_IF
	ELSE
		Mach_Control.DT_b.Error[8]:=TRUE;//叠正极片凸轮耦合时，正极片不在取片位
		DP_Step0:=10001;
	END_IF	
	
1150://纠偏台回初始位
	//纠偏平台X1移动至初始位
	IF NOT DP_SinStepe THEN
		IF arrAxisCtrl[AxiseNo.AxisName.AndeviationX1].Status.Homed  AND arrAxisCtrl[AxiseNo.AxisName.AndeviationX1].Status.NoMoving AND NOT  arrAxisCtrl[AxiseNo.AxisName.AndeviationX1].Status.Error THEN
			IF arrAxisCtrl[AxiseNo.AxisName.AndeviationX1].Cmd.arrbRealPoint[1] THEN
				arrAxisCtrl[AxiseNo.AxisName.AndeviationX1].Cmd.iGoSetPos:=0;
			ELSE
				arrAxisCtrl[AxiseNo.AxisName.AndeviationX1].Cmd.iGoSetPos:=1;
			END_IF					
		END_IF
		//纠偏平台X2移动至初始位
		IF arrAxisCtrl[AxiseNo.AxisName.AndeviationX2].Status.Homed  AND arrAxisCtrl[AxiseNo.AxisName.AndeviationX2].Status.NoMoving AND NOT  arrAxisCtrl[AxiseNo.AxisName.AndeviationX2].Status.Error THEN
			IF arrAxisCtrl[AxiseNo.AxisName.AndeviationX2].Cmd.arrbRealPoint[1] THEN
				arrAxisCtrl[AxiseNo.AxisName.AndeviationX2].Cmd.iGoSetPos:=0;
			ELSE
				arrAxisCtrl[AxiseNo.AxisName.AndeviationX2].Cmd.iGoSetPos:=1;
			END_IF					
		END_IF
		//纠偏平台X2移动至初始位
		IF arrAxisCtrl[AxiseNo.AxisName.AndeviationY].Status.Homed  AND arrAxisCtrl[AxiseNo.AxisName.AndeviationY].Status.NoMoving AND NOT  arrAxisCtrl[AxiseNo.AxisName.AndeviationY].Status.Error THEN
			IF arrAxisCtrl[AxiseNo.AxisName.AndeviationY].Cmd.arrbRealPoint[1] THEN
				arrAxisCtrl[AxiseNo.AxisName.AndeviationY].Cmd.iGoSetPos:=0;
			ELSE
				arrAxisCtrl[AxiseNo.AxisName.AndeviationY].Cmd.iGoSetPos:=1;
			END_IF					
		END_IF
		IF arrAxisCtrl[AxiseNo.AxisName.AndeviationX1].Cmd.arrbRealPoint[1] AND arrAxisCtrl[AxiseNo.AxisName.AndeviationX2].Cmd.arrbRealPoint[1] AND arrAxisCtrl[AxiseNo.AxisName.AndeviationY].Cmd.arrbRealPoint[1] THEN
			DT_SingeMode();//单步选择	
			DP_Step0:=1200;	
			DT_TON[5].IN:=FALSE;
		END_IF	
	END_IF
1200:
	IF NOT DP_SinStepe THEN
		IF arrAxisCtrl[AxiseNo.AxisName.AnDTCarryingUpDown].Cmd.arrbRealPoint[3] THEN
			arrAxisCtrl[AxiseNo.AxisName.AnDTCarryingUpDown].Cmd.iGoSetPos:=0;
			/// 吸盘破真空    纠偏台开真空
			arrCyCtrl[arrCyNo.ElectValveName.AnDTCarryingVacuum].Cmd.bON:=TRUE;	//正极叠台搬运升降真空	真空
			arrCyCtrl[arrCyNo.ElectValveName.AnDTCarryingVacuum].Cmd.bOFF:=FALSE;	//正极叠台搬运升降真空破真空		
			arrCyCtrl[arrCyNo.ElectValveName.AnDTCarryingVacuumBark].Cmd.bON:=TRUE;	//正极叠台搬运升降真空	真空
			arrCyCtrl[arrCyNo.ElectValveName.AnDTCarryingVacuumBark].Cmd.bOFF:=FALSE;	//正极叠台搬运升降真空破真空											
			arrCyCtrl[arrCyNo.ElectValveName.AndeviationVacuum].Cmd.bON:=TRUE;	//正极纠偏台真空			
			arrCyCtrl[arrCyNo.ElectValveName.AndeviationVacuum].Cmd.bOFF:=FALSE;	//正极纠偏台真空	
			DT_SingeMode();//单步选择	
			DP_Step0:=1250;
			DT_TON[5].IN:=TRUE;
		ELSE
			arrAxisCtrl[AxiseNo.AxisName.AnDTCarryingUpDown].Cmd.iGoSetPos:=3;//负极搬运升降2上升至凸轮耦合初始高度
		END_IF	
	END_IF	
1250://叠台搬运极片放回纠偏台
	IF NOT DP_SinStepe THEN
		  IF DT_TON[5].Q THEN
				IF arrAxisCtrl[AxiseNo.AxisName.AnDTCarryingUpDown].Cmd.arrbRealPoint[4] THEN
					arrAxisCtrl[AxiseNo.AxisName.AnDTCarryingUpDown].Cmd.iGoSetPos:=0;
					/// 吸盘破真空    纠偏台开真空
					Mach_Control.An_b.An_deviationFalg:=TRUE;//复位纠偏平台有料标记
					Mach_Control.An_b.An_DPCarryingFalg:=FALSE;//负极搬运真空吸盘有料标记复位
					Par.stDT_date.An_MQ_Slice[1]:=Par.stDT_date.An_MQ_Slice[2];
					DT_SingeMode();//单步选择	
					DP_Step0:=1300;
					DT_TON[5].IN:=FALSE;
				ELSE
					arrAxisCtrl[AxiseNo.AxisName.AnDTCarryingUpDown].Cmd.iGoSetPos:=4;//负极搬运升降2上升至凸轮耦合初始高度
				END_IF	
		 END_IF		
	END_IF			
1300:
	DP_Step0:=2000;	
	

	
	
	
